// TwinCAT 3 PLC project MPM_PUMP
// ProgramVersion: 3.1.4024.0
// libraries:
//   MPM_FBResult, * (MatrixPM)
//   MPM_JsonParser, * (MatixPM)
//   Tc2_MC2, * (Beckhoff Automation GmbH)
//   Tc2_Standard, * (Beckhoff Automation GmbH)
//   Tc2_System, * (Beckhoff Automation GmbH)
//   Tc2_Utilities, * (Beckhoff Automation GmbH)
//   Tc3_IotBase, * (Beckhoff Automation GmbH)
//   Tc3_Module, * (Beckhoff Automation GmbH)
// project tree:
//   / Class Diagram.TcCD (not stored), PlcTask.TcTTO
//   FBs/Abstracts/ FB_AxisControl.TcPOU, FB_ConfigBase.TcPOU, FB_DiscreteEvents.TcPOU, FB_EventScheduler.TcPOU, FB_PackMLControl.TcPOU, FB_TimeEvents.TcPOU
//   FBs/ FB_EventArray.TcPOU, FB_Kinenmatics.TcPOU, FB_Kinenmatics_V2.TcPOU
//   FBs/IO_Mapping/ FB_IOMappingJson.TcPOU (excluded from build)
//   FBs/IO_Mapping/TcCom/ FB_IOMapping.TcPOU (excluded from build)
//   FBs/IO_Mapping/Types/ ST_IOMappingJson_OLD.TcDUT, ST_IOMappingJson.TcDUT
//   FBs/JSON/ FB_NCAxisJson.TcPOU, FB_NCAxisJson_V2.TcPOU, FB_ValuesJson.TcPOU, ST_AxisMap.TcDUT, ST_AxisMapping.TcDUT
//   FBs/Main/ E_PackMLStates.TcDUT, FB_JsonFile.TcPOU, FB_PackMLControl_Auto.TcPOU, FB_Pump.TcPOU, FB_Squeegee.TcPOU
//   FBs/System/ FB_ConfigControl.TcPOU
//   FUN/ F_Add1.TcPOU, F_INIT_ST_AnyType.TcPOU
//   POUs/ MAIN.TcPOU
// real-time tasks:
//   TASK PlcTask: cycle T#10ms, priority 20, ADS port 350
// motion (NC):
//   TASK NC-Task 1 SAF: cycle T#2ms, priority 4, ADS port 501
//   TASK NC-Task 1 SVB: cycle T#10ms, priority 8, ADS port 511
//   AXIS Axis 1 (id 1)
//     General: UnitName=°
//     Dynamic: Acceleration=5355.76, Deceleration=5355.76, Jerk=16067.3
//     Velo: RefSearch=35.70505, RefSync=35.70505, SlowManual=178.52525, FastManual=1071.1515, Fast=3570.505, Maximum=3570.51
//     OtherSettings: AllowMotionCmdToSlave=true
//     encoder EncType=1
//       EncPara: ScaleFactorNumerator=360, ScaleFactorDenominator=4194304
//     drive DrvType=5
//       Analog: VeloReferenz=3927.5555, TorqueSetpointScale=10, ScaleFactorActTorque=0.1
//       TimeComp: TaskDelayCycles=1
//     controller CtrType=1
//       CtrPara: PriorControlFactor=1
//         Observer: BandWidth=20
// I/O:
//   DEVICE Device 1 (EtherCAT) (disabled), AmsNetId 5.125.204.206.2.1
//     Term 1 (EK1200) [EK1200-5000 EtherCAT Power supply (2A E-Bus)]
//       Term 2 (EL6224) [EL6224 (IO Link Master)]
//       Term 3 (EL1904) [EL1904, 4 Ch. Safety Input 24V, TwinSAFE]
//         modules: Module 1 (FSOES)
//       Term 4 (EL9011) [EL9011 End Terminal]
//   DEVICE Device 2 (EtherCAT) (disabled), AmsNetId 5.125.204.206.3.1
//     Drive 5 (AX5206-0000-0214) [AX5206-0000-0214 EtherCAT Drive (SoE, 2 Ch.)]
// variable links:
//   MPM_PUMP/MPM_PUMP Instance <-> NC-Task 1 SAF/Axes/Axis 1
//     PlcTask Inputs/MAIN.fbPump.axis.NcToPlc <-> Outputs/ToPlc
//     PlcTask Outputs/MAIN.fbPump.axis.PlcToNc <-> Inputs/FromPlc

CONFIGURATION MPM_PUMP
    RESOURCE PLC ON TwinCAT3
        TASK PlcTask(INTERVAL := T#10ms, PRIORITY := 20);
        PROGRAM MAIN WITH PlcTask : MAIN;
    END_RESOURCE
END_CONFIGURATION

// ---- FBs/IO_Mapping/Types/ST_IOMappingJson_OLD.TcDUT
TYPE ST_IOMappingJson_OLD :
STRUCT
	name : STRING;
	deviceNum : WORD;
	channel : USINT;
	ethercatDeviceNum : WORD;
	ioLinkDevice : USINT;
	ioLinkSlaveChannel : USINT;	
	pAny : MPM_JsonParser.ST_AnyType_User;
END_STRUCT
END_TYPE

// ---- FBs/IO_Mapping/Types/ST_IOMappingJson.TcDUT
TYPE ST_IOMappingJson :
STRUCT
	name : STRING;
	deviceNum : WORD;
	channel : USINT;
	ethercatDeviceNum : WORD;
	ioLinkDevice : USINT;
	ioLinkSlaveChannel : USINT;	
	pAny : MPM_JsonParser.ST_AnyType_User;
END_STRUCT
END_TYPE

// ---- FBs/JSON/ST_AxisMap.TcDUT
TYPE ST_AxisMap :
STRUCT
	stAxisMappingJson : ARRAY [0..67] OF  ST_AxisMapping;	
END_STRUCT
END_TYPE

// ---- FBs/JSON/ST_AxisMapping.TcDUT
TYPE ST_AxisMapping :
STRUCT
	name : STRING;
	indexOffset : UDINT;
	pAny : MPM_JsonParser.ST_AnyType_User;
END_STRUCT
END_TYPE

// ---- FBs/Main/E_PackMLStates.TcDUT
{attribute 'qualified_only'}
{attribute 'strict'}
TYPE E_PackMLStates :
(
	idle,
	starting,
	execute,
	completing,
	complete,
	suspdending,
	suspended,
	un_suspsending,
	holding,
	held,
	un_holding,
	aborting,
	aborted,
	stopping,
	stopped
);
END_TYPE

// ---- POUs/MAIN.TcPOU
PROGRAM MAIN
VAR
	ap_fbEvents : ARRAY [0..1023] OF POINTER TO FB_DiscreteEvents; //All assest events combinded
	index : UDINT;
	//machine assets
	fbPump : FB_Pump('fbName');
	fbPump1 : FB_Pump('fbName1');
	fbPump2 : FB_Pump('fbName2');	
	fbPump3 : FB_Pump('fbName3');	
	a_pFBConfigJson : ARRAY [0..3] OF POINTER TO FB_ConfigBase;

	//config control
	fbConfigControl : FB_ConfigControl;
	fbConfigControl_JsonRecipeResult : HRESULT;
	fbConfigControl_JsonSystemResult : HRESULT;
	fbConfigControl_JsonIOResult : HRESULT;
	fbConfigControl_JsonAxisResult : HRESULT;	
	jsonRecipeDoc : STRING(10000);
	jsonSystemDoc : STRING(50000);
	jsonIODoc : STRING(50000);
	jsonAxisDoc : STRING(50000);
	
	//stateMachine
	fbPackMLControlAuto : FB_PackMLControl_Auto; 
	//Node-Red
	fbJsonMQTT : Tc3_IotBase.FB_IotMqttClient;
	mqttPubRate : TON;

END_VAR
//temp 
VAR
	pPointer : ARRAY [0..10] OF POINTER TO MPM_JsonParser.ST_AnyType_User;
	sizeOfValue : DINT;
	position : LREAL;
	dynamicMem : ARRAY [0..65354] OF PVOID;	
	fbKinenmatics : FB_Kinenmatics;
	fbKinenmatics2 : FB_Kinenmatics_V2;	
END_VAR
//Event Test
VAR
x : DINT;
y : DINT;
aLreal : ARRAY [0..0] OF LREAL;
fbPump_OpenValve_Result : HResult := 1;
fbPump_CloseValve_Result : HResult := 1;
fbPump_EnablePump : HResult := 1;
fbPump_HomePump : HResult := 1;
fbPump_MoveAbs : HResult := 1;
fbPump_MoveIncerment : HResult := 1;
fbPump_MoveHalt : HResult := 1;
END_VAR



A_INIT();
A_ConfigControl();
A_Events();

fbPackMLControlAuto.ap_fbEvents := ADR(ap_fbEvents);
fbPackMLControlAuto.M_ExecuteControl();

ACTION A_ConfigControl:


fbConfigControl.a_pFBConfigJson := ADR(a_pFBConfigJson);
fbConfigControl.ua_pFBConfigJson := SIZEOF(a_pFBConfigJson); //Mapping machine assest
//Set json files
fbConfigControl.M_SetJsonRecipe(fbConfigControl_JsonRecipeResult,jsonRecipeDoc);
fbConfigControl.M_SetJsonSystem(fbConfigControl_JsonSystemResult,jsonSystemDoc);
fbConfigControl.M_SetJsonIO(fbConfigControl_JsonIOResult,jsonIODoc);
fbConfigControl.M_SetJsonAxis(fbConfigControl_JsonAxisResult,jsonAxisDoc);
//fbConfigControl_JsonRecipeResult := fbConfigControl.M_GetJsonRecipe(fbConfigControl_JsonRecipeResult,jsonRecipeDoc);


fbJsonMQTT.Execute(TRUE);
mqttPubRate(in := fbJsonMQTT.bConnected, PT := T#500MS);
IF mqttPubRate.Q AND_THEN fbJsonMQTT.Publish('axis',ADR(jsonAxisDoc),LEN2(ADR(jsonAxisDoc)),0,FALSE,FALSE) THEN
	mqttPubRate(in := FALSE);
END_IF
END_ACTION

ACTION A_Events:
fbPump.M_Execute();
fbPump_OpenValve_Result := fbPump.M_Events(fbPump_OpenValve_Result,1);
fbPump_CloseValve_Result := fbPump.M_Events(fbPump_CloseValve_Result,2);
fbPump_EnablePump := fbPump.fbEventEnable.M_Execute(fbPump_EnablePump);
fbPump_HomePump := fbPump.fbEventHomePump.M_Execute(fbPump_HomePump,);
fbPump_MoveIncerment := fbPump.fbEventPumpInterminate.M_Execute(fbPump_MoveIncerment);
fbPump_MoveHalt := fbPump.fbEventMoveHalt.M_Execute(fbPump_MoveHalt);
FOR x := 0 TO 4 BY 1 DO
	fbPump.fbEventMoveAbs.F_GetAnyType(x,p => pPointer[0]);
	F_INIT_ST_AnyType(pPointer[0]);
END_FOR	
fbPump_MoveAbs := fbPump.M_Events(fbPump_MoveAbs,5);

IF fbPump_OpenValve_Result = E_Result.S_OK THEN
	fbPump_OpenValve_Result := E_Result.S_DONE;
END_IF
IF fbPump_CloseValve_Result = E_Result.S_OK THEN
	fbPump_CloseValve_Result := E_Result.S_DONE;
END_IF
IF fbPump_EnablePump = E_Result.S_OK THEN
	fbPump_EnablePump := E_Result.S_DONE;
END_IF
IF fbPump_HomePump = E_Result.S_OK THEN
	fbPump_HomePump := E_Result.S_DONE;
END_IF 
IF fbPump_MoveAbs = E_Result.S_OK THEN
	fbPump_MoveAbs := E_Result.S_DONE;
END_IF 
IF fbPump_MoveIncerment = E_Result.S_OK THEN
	fbPump_MoveIncerment := E_Result.S_DONE;
END_IF 
IF fbPump_MoveHalt = E_Result.S_OK THEN
	fbPump_MoveHalt := E_Result.S_DONE;
END_IF
END_ACTION

ACTION A_INIT:


//Map all 
IF index = 0 THEN
	a_pFBConfigJson[0] := ADR(fbPump);
	a_pFBConfigJson[1] := ADR(fbPump1);
	a_pFBConfigJson[2] := ADR(fbPump2);
	a_pFBConfigJson[3] := ADR(fbPump3);	
	
	FOR x := 0 TO 3 BY 1 DO
		FOR y := 0 TO a_pFBConfigJson[x]^.P_GetNumOfEvents - 1 BY 1 DO
			IF a_pFBConfigJson[x]^.M_GetEvent(ADR(ap_fbEvents[index]),y) = E_Result.S_OK THEN
				index := index + 1;	
			ELSE
				CONTINUE;
			END_IF	
		END_FOR
	END_FOR
END_IF
END_ACTION

END_PROGRAM

// ---- FBs/Abstracts/FB_DiscreteEvents.TcPOU
(*
Standard way to set up events to be tied to other parts of the project. might make an interface
*)
{attribute 'reflection'} 
FUNCTION_BLOCK FB_DiscreteEvents
VAR_INPUT
END_VAR
VAR_OUTPUT
END_VAR
VAR
	pstAnyType_User : POINTER TO MPM_JsonParser.ST_AnyType_User; //array 
	uAnyType_User : DINT; //Len of array 
	pfbConfigBase : POINTER TO FB_ConfigBase; 
	eventID : DINT;
    {attribute 'instance-path'} 
    {attribute 'noinit'}	
	_eventName : STRING(1024);
END_VAR
VAR CONSTANT
	sizeOfAnyType_User : DINT := SIZEOF(MPM_JsonParser.ST_AnyType_User);
END_VAR

METHOD PUBLIC F_GetAnyType : HResult
VAR_INPUT
	arrayPosition : DINT;
END_VAR
VAR_OUTPUT
	p : POINTER TO MPM_JsonParser.ST_AnyType_User;
END_VAR
VAR
	pointerOffset : DINT;
END_VAR
IF pstAnyType_User = 0 THEN // no values
	F_GetAnyType := MPM_FBResult.E_Result.S_FAILED;
END_IF
F_GetAnyType := pfbConfigBase^.F_GetArrayPosition(uAnyType_User,sizeOfAnyType_User,arrayPosition,offset => pointerOffset);
IF F_GetAnyType = MPM_FBResult.E_Result.S_OK THEN
	p := pstAnyType_User + pointerOffset;
ELSE
	F_GetAnyType := MPM_FBResult.E_Result.S_FAILED;
END_IF
END_METHOD

METHOD FB_exit : BOOL
VAR_INPUT
	bInCopyCode : BOOL; // if TRUE, the exit method is called for exiting an instance that is copied afterwards (online change).
END_VAR

VAR
	pstAnyType_User : POINTER TO MPM_JsonParser.ST_AnyType_User; //array 
	length : DINT; 
	offset : DINT;
	x : DINT;
	pByte : POINTER TO BYTE;
END_VAR
IF bInCopyCode = FALSE THEN
	IF pfbConfigBase^.F_GetArrayLength(uAnyType_User,sizeOfAnyType_User, length => length) = MPM_FBResult.E_Result.S_OK THEN
		FOR x := 0 TO length BY 1 DO
			pfbConfigBase^.F_GetArrayPosition(uAnyType_User,sizeOfAnyType_User,x,offset => offset);
			pstAnyType_User := THIS^.pstAnyType_User + offset;
			pByte := pstAnyType_User^.pvalue;
			__DELETE(pByte);
		END_FOR
	END_IF
END_IF
END_METHOD

METHOD FB_init : BOOL
VAR_INPUT
	bInitRetains : BOOL; // if TRUE, the retain variables are initialized (warm start / cold start)
	bInCopyCode : BOOL;  // if TRUE, the instance afterwards gets moved into the copy code (online change)
	pfbConfigBase : POINTER TO FB_ConfigBase; 
	eventID : DINT;
	pstAnyType_User : POINTER TO MPM_JsonParser.ST_AnyType_User; //array 
	uAnyType_User : DINT; //Len of array 	
END_VAR
THIS^.pfbConfigBase := pfbConfigBase;
THIS^.pstAnyType_User := pstAnyType_User;
THIS^.uAnyType_User := uAnyType_User;
THIS^.eventID := eventID;
END_METHOD

METHOD PUBLIC M_Execute : HRESULT
VAR_INPUT
	lastResult : HResult;
END_VAR
IF pfbConfigBase > 0 THEN 
	M_Execute := pfbConfigBase^.M_Events(lastResult,eventID);
END_IF
END_METHOD

PROPERTY PUBLIC P_EventId : Dint
GET
END_GET
END_PROPERTY

PROPERTY PUBLIC P_EventName : String(1024)
GET
P_EventName := _eventName;
END_GET
END_PROPERTY

END_FUNCTION_BLOCK

// ---- FBs/Abstracts/FB_ConfigBase.TcPOU
(*
Will be an abstract class that will be used to configure all parts of the machine through json
*)

FUNCTION_BLOCK ABSTRACT FB_ConfigBase
VAR_INPUT
END_VAR
VAR_OUTPUT
END_VAR
VAR 
	_fbName : STRING; //name of FB set on init
END_VAR

METHOD _F_Axis : HRESULT
VAR_IN_OUT
	a_pstAxisParameterSet : POINTER TO Tc2_MC2.ST_AxisParameterSet; //pointer to array
	pstAxisMapping : UDINT;
END_VAR
END_METHOD

METHOD PROTECTED ABSTRACT _F_IO : HResult
VAR_IN_OUT
	a_pstIOMappingJson : POINTER TO ST_IOMappingJson; //pointer to array
	ustIOMappingJson : UDINT; 		
END_VAR
END_METHOD

(*
return the list of vars that want to be saved and loaded 
*)

METHOD PROTECTED ABSTRACT _F_Recipe : HResult
VAR_IN_OUT
	a_pstAnyTypeUser : POINTER TO MPM_JsonParser.ST_AnyType_User; //pointer to array
	uAnyTypeUser : UDINT; //size of array	
END_VAR
VAR_OUTPUT

END_VAR
END_METHOD

METHOD PROTECTED ABSTRACT _F_System : HResult
VAR_IN_OUT
	a_pstAnyTypeUser : POINTER TO MPM_JsonParser.ST_AnyType_User; //pointer to array
	uAnyTypeUser : UDINT; //size of array	
END_VAR
END_METHOD

METHOD PUBLIC FINAL F_AXIS : HRESULT
VAR_INPUT
	lastResult : HRESULT;
	sJson : SJsonValue;
	pfbJsonSchema : POINTER TO FB_NCAxisJson_V2;	
	bGet : BOOL;
END_VAR

VAR_INST
	_fbResult : FB_ResultHelper_V2;
	pResult : POINTER TO HRESULT;
END_VAR

VAR
	a_pstAxisParameterSet : POINTER TO Tc2_MC2.ST_AxisParameterSet;
	dstAxisParameterSet : UDINT; //number of bytes in a_stAnyUser
	
	uSizeOfArray : UDINT;
	
	pstAxisParameterSet : POINTER TO Tc2_MC2.ST_AxisParameterSet; //pointer for loop
	x : UDINT;
END_VAR


VAR CONSTANT
	uSizeOfStAnyType : UDINT := SIZEOF(Tc2_MC2.ST_AxisParameterSet);
END_VAR
IF _fbResult.M_MethodResult(F_AXIS,ADR(pResult),lastResult) = FALSE THEN
	RETURN;
END_IF


pResult^ := _F_Axis(a_pstAxisParameterSet,dstAxisParameterSet);
//pResult^ := MPM_FBResult.E_Result.S_WORKING;
IF bGet = FALSE THEN
	sJson := pfbJsonSchema^.M_SetJsonMember(sJson,_fbName);
	IF a_pstAxisParameterSet > 0 AND dstAxisParameterSet > 0 AND uSizeOfStAnyType > 0 THEN //make sure all values are vaild
		uSizeOfArray := dstAxisParameterSet/uSizeOfStAnyType - 1; //get number of items in array
		FOR x := 0 TO uSizeOfArray BY 1 DO //loop through all items 
			pstAxisParameterSet := a_pstAxisParameterSet + uSizeOfStAnyType*x; // get array position
			pResult^ := pfbJsonSchema^.M_SetAxisJson(pResult^,sJson,pstAxisParameterSet);
		END_FOR
	END_IF	
ELSIF bGet = TRUE THEN
	sJson := pfbJsonSchema^.FindMember(sJson,_fbName);
	IF a_pstAxisParameterSet > 0 AND dstAxisParameterSet > 0 AND uSizeOfStAnyType > 0 THEN //make sure all values are vaild
		uSizeOfArray := dstAxisParameterSet/uSizeOfStAnyType - 1; //get number of items in array
		FOR x := 0 TO uSizeOfArray BY 1 DO //loop through all items 
			pstAxisParameterSet := a_pstAxisParameterSet + uSizeOfStAnyType*x; // get array position
			pResult^ := pfbJsonSchema^.M_GetAxisJson(pResult^,sJson,pstAxisParameterSet);
		END_FOR
	END_IF
END_IF
END_METHOD

METHOD PROTECTED F_Event_ST_AnyType_Compare : HResult
VAR_INPUT
	srcvar : POINTER TO MPM_JsonParser.ST_AnyType_User; //PVOID FOR any value
	desvar : POINTER TO MPM_JsonParser.ST_AnyType_User;	//What was input
END_VAR
VAR
END_VAR
IF srcvar^.typeclass = desvar^.typeclass AND srcvar^.diSize = desvar^.diSize THEN
	desvar^.pvalue := srcvar^.pvalue;
	F_Event_ST_AnyType_Compare := MPM_FBResult.E_Result.S_OK;
ELSE
	F_Event_ST_AnyType_Compare := MPM_FBResult.E_Result.S_FAILED;	
END_IF
END_METHOD

METHOD PUBLIC F_GetArrayLength : HResult
VAR_INPUT
	sizeOfInst : DINT;
	sizeOFType : DINT;
END_VAR
VAR_OUTPUT
	length : DINT;
END_VAR
VAR
	_numOfElements : DINT;
END_VAR
IF sizeOFType > 0 AND sizeOfInst > 0 THEN
	_numOfElements := sizeOfInst/sizeOFType -1;
	IF _numOfElements > 0 THEN
		length := _numOfElements;
		F_GetArrayLength := MPM_FBResult.E_Result.S_OK;
	END_IF
ELSE
	F_GetArrayLength := MPM_FBResult.E_Result.S_FAILED;
	RETURN;
END_IF
END_METHOD

METHOD PUBLIC F_GetArrayPosition : HResult
VAR_INPUT
	sizeOfInst : DINT;
	sizeOFType : DINT;
	index : DINT;
END_VAR
VAR_OUTPUT
	offset : DINT;
	length : DINT;
END_VAR
VAR
END_VAR
F_GetArrayPosition := F_GetArrayLength(sizeOfInst,sizeOFType, length => length);
IF F_GetArrayPosition = MPM_FBResult.E_Result.S_OK THEN
	IF index >= 0 AND index <= length THEN
		offset := sizeOFType*index;
	ELSE
		F_GetArrayPosition := MPM_FBResult.E_Result.S_FAILED;
	END_IF
ELSE
	F_GetArrayPosition := MPM_FBResult.E_Result.S_OK;
END_IF
END_METHOD

METHOD PUBLIC FINAL F_IO : HRESULT
VAR_INPUT
	lastResult : HRESULT;
	sJson : SJsonValue;
	pfbJsonSchema : POINTER TO FB_JsonSchemaEx_OLD;
	bGet : BOOL;	
END_VAR

VAR_INST
	_fbResult : FB_ResultHelper_V2;
	pResult : POINTER TO HRESULT;
END_VAR

VAR
	a_pstIOMappingJson : POINTER TO ST_IOMappingJson; // pointer to array of vars
	uAnyTypeUser : UDINT; //number of bytes in a_stAnyUser
	
	uSizeOfArray : UDINT;
	pstIOMappingJson : POINTER TO ST_IOMappingJson; //pointer for loop
	x : UDINT;
END_VAR


VAR CONSTANT
	uSizeOfStAnyType : UDINT := SIZEOF(ST_IOMappingJson);
END_VAR
IF _fbResult.M_MethodResult(F_IO,ADR(pResult),lastResult) = FALSE THEN
	RETURN;
END_IF


pResult^ := _F_IO(a_pstIOMappingJson,uAnyTypeUser); //gets pointer from FB


pResult^ := MPM_FBResult.E_Result.S_WORKING;
//set
IF bGet = FALSE THEN
	sJson := pfbJsonSchema^.M_SetJsonMember(sJson,_fbName);
	IF a_pstIOMappingJson > 0 AND_THEN uAnyTypeUser > 0 AND uSizeOfStAnyType > 0 THEN //make sure all values are vaild
		uSizeOfArray := uAnyTypeUser/uSizeOfStAnyType - 1; //get number of items in array
		FOR x := 0 TO uSizeOfArray BY 1 DO //loop through all items 
			pstIOMappingJson := a_pstIOMappingJson + uSizeOfStAnyType*x; // get array position
			sJson := pfbJsonSchema^.M_SetJsonMember(sJson,pstIOMappingJson^.name); //set json value
			pfbJsonSchema^.M_SetJsonMemberValue(sJson,'deviceNum',pstIOMappingJson^.deviceNum); //set json value			
			pfbJsonSchema^.M_SetJsonMemberValue(sJson,'channel',pstIOMappingJson^.channel); //set json value
			//IO-link
			pfbJsonSchema^.M_SetJsonMemberValue(sJson,'ethercatDeviceNum',pstIOMappingJson^.ethercatDeviceNum); //set json value
			pfbJsonSchema^.M_SetJsonMemberValue(sJson,'ioLinkDevice',pstIOMappingJson^.ioLinkDevice); //set json value
			pfbJsonSchema^.M_SetJsonMemberValue(sJson,'ioLinkSlaveChannel',pstIOMappingJson^.ioLinkSlaveChannel); //set json value
		END_FOR
		pResult^ := MPM_FBResult.E_Result.S_OK;
	ELSE
		pResult^ := MPM_FBResult.E_Result.S_FAILED;
	END_IF
//get
ELSIF bGet = TRUE THEN
	sJson := pfbJsonSchema^.FindMember(sJson,_fbName);
	IF a_pstIOMappingJson > 0 AND_THEN uAnyTypeUser > 0 AND uSizeOfStAnyType > 0 THEN //make sure all values are vaild
		uSizeOfArray := uAnyTypeUser/uSizeOfStAnyType - 1; //get number of items in array
		FOR x := 0 TO uSizeOfArray BY 1 DO //loop through all items 
			pstIOMappingJson := a_pstIOMappingJson + uSizeOfStAnyType*x; // get array position
			sJson := pfbJsonSchema^.M_SetJsonMember(sJson,pstIOMappingJson^.name); //set json value
			pfbJsonSchema^.M_GetJsonMemberValue(sJson,'channel',pstIOMappingJson^.channel); //set json value
			pfbJsonSchema^.M_GetJsonMemberValue(sJson,'deviceNum',pstIOMappingJson^.deviceNum); //set json value
			pfbJsonSchema^.M_GetJsonMemberValue(sJson,'ethercatDeviceNum',pstIOMappingJson^.ethercatDeviceNum); //set json value
			pfbJsonSchema^.M_GetJsonMemberValue(sJson,'ioLinkDevice',pstIOMappingJson^.ioLinkDevice); //set json value
			pfbJsonSchema^.M_GetJsonMemberValue(sJson,'ioLinkSlaveChannel',pstIOMappingJson^.ioLinkSlaveChannel); //set json value
		END_FOR
		pResult^ := MPM_FBResult.E_Result.S_OK;
	ELSE
		pResult^ := MPM_FBResult.E_Result.S_FAILED;
	END_IF
END_IF
END_METHOD

METHOD PROTECTED F_Map_ST_IOMappingJson : HRESULT
VAR_INPUT
	stIOMappingJson : POINTER TO ST_IOMappingJson;
	name : STRING;
	pPVoid : POINTER TO PVOID;
END_VAR
END_METHOD

METHOD PUBLIC FINAL F_Recipe : HRESULT
VAR_INPUT
	lastResult : HRESULT;
	sJson : SJsonValue;
	pfbJsonSchema : POINTER TO FB_JsonSchemaEx_OLD;	
	bGet : BOOL;
END_VAR

VAR_INST
	_fbResult : FB_ResultHelper_V2;
	pResult : POINTER TO HRESULT;
END_VAR

VAR
	a_stAnyUser : POINTER TO MPM_JsonParser.ST_AnyType_User; // pointer to array of vars
	uAnyTypeUser : UDINT; //number of bytes in a_stAnyUser
	
	uSizeOfArray : UDINT;
	pstAnyUser : POINTER TO MPM_JsonParser.ST_AnyType_User; //pointer for loop
	x : UDINT;
END_VAR

VAR CONSTANT
	uSizeOfStAnyType : UDINT := SIZEOF(MPM_JsonParser.ST_AnyType_User);
END_VAR
IF _fbResult.M_MethodResult(F_Recipe,ADR(pResult),lastResult) = FALSE THEN
	RETURN;
END_IF


pResult^ := _F_Recipe(a_stAnyUser,uAnyTypeUser);


pResult^ := MPM_FBResult.E_Result.S_WORKING;

//set
IF bGet = FALSE THEN
	sJson := pfbJsonSchema^.M_SetJsonMember(sJson,_fbName);
	IF a_stAnyUser > 0 AND_THEN uAnyTypeUser > 0 AND uSizeOfStAnyType > 0 THEN //make sure all values are vaild
		uSizeOfArray := uAnyTypeUser/uSizeOfStAnyType - 1; //get number of items in array
		FOR x := 0 TO uSizeOfArray BY 1 DO //loop through all items 
			pstAnyUser := a_stAnyUser + uSizeOfStAnyType*x; // get array position
				pfbJsonSchema^.M_SetJsonMemberValue_AnyType(sJson,pstAnyUser^.name,pstAnyUser^); //set json value
		END_FOR
		pResult^ := MPM_FBResult.E_Result.S_OK;
	ELSE
		pResult^ := MPM_FBResult.E_Result.S_FAILED;
	END_IF
	
//get
ELSIF bGet = TRUE THEN 	
	sJson := pfbJsonSchema^.FindMember(sJson,_fbName);
	IF a_stAnyUser > 0 AND_THEN uAnyTypeUser > 0 AND uSizeOfStAnyType > 0 THEN //make sure all values are vaild
		uSizeOfArray := uAnyTypeUser/uSizeOfStAnyType - 1; //get number of items in array
		FOR x := 0 TO uSizeOfArray BY 1 DO //loop through all items 
			pstAnyUser := a_stAnyUser + uSizeOfStAnyType*x; // get array position
				pfbJsonSchema^.M_GetJsonMemberValue_AnyType(sJson,pstAnyUser^.name,pstAnyUser^); //set json value
		END_FOR
		pResult^ := MPM_FBResult.E_Result.S_OK;
	ELSE
		pResult^ := MPM_FBResult.E_Result.S_FAILED;
	END_IF
END_IF
END_METHOD

METHOD PUBLIC FINAL F_System : HRESULT
VAR_INPUT
	lastResult : HRESULT;
	sJson : SJsonValue;
	pfbJsonSchema : POINTER TO FB_JsonSchemaEx_OLD;	
	bGet : BOOL;	
END_VAR

VAR_INST
	_fbResult : FB_ResultHelper_V2;
	pResult : POINTER TO HRESULT;
END_VAR

VAR
	a_stAnyUser : POINTER TO MPM_JsonParser.ST_AnyType_User; // pointer to array of vars
	uAnyTypeUser : UDINT; //number of bytes in a_stAnyUser
	
	uSizeOfArray : UDINT;
	pstAnyUser : POINTER TO MPM_JsonParser.ST_AnyType_User; //pointer for loop
	x : UDINT;
END_VAR


VAR CONSTANT
	uSizeOfStAnyType : UDINT := SIZEOF(MPM_JsonParser.ST_AnyType_User);
END_VAR
IF _fbResult.M_MethodResult(F_System,ADR(pResult),lastResult) = FALSE THEN
	RETURN;
END_IF


pResult^ := _F_System(a_stAnyUser,uAnyTypeUser);
//set
IF bGet = FALSE THEN
	pResult^ := MPM_FBResult.E_Result.S_WORKING;
	sJson := pfbJsonSchema^.M_SetJsonMember(sJson,_fbName);
	IF a_stAnyUser > 0 AND_THEN uAnyTypeUser > 0 AND uSizeOfStAnyType > 0 THEN //make sure all values are vaild
		uSizeOfArray := uAnyTypeUser/uSizeOfStAnyType - 1; //get number of items in array
		FOR x := 0 TO uSizeOfArray BY 1 DO //loop through all items 
			pstAnyUser := a_stAnyUser + uSizeOfStAnyType*x; // get array position
				pfbJsonSchema^.M_SetJsonMemberValue_AnyType(sJson,pstAnyUser^.name,pstAnyUser^); //set json value
		END_FOR
		pResult^ := MPM_FBResult.E_Result.S_OK;
	ELSE
		pResult^ := MPM_FBResult.E_Result.S_FAILED;
	END_IF

//get	
ELSIF bGet = TRUE THEN
	sJson := pfbJsonSchema^.FindMember(sJson,_fbName);
	IF a_stAnyUser > 0 AND_THEN uAnyTypeUser > 0 AND uSizeOfStAnyType > 0 THEN //make sure all values are vaild
		uSizeOfArray := uAnyTypeUser/uSizeOfStAnyType - 1; //get number of items in array
		FOR x := 0 TO uSizeOfArray BY 1 DO //loop through all items 
			pstAnyUser := a_stAnyUser + uSizeOfStAnyType*x; // get array position
				pfbJsonSchema^.M_GetJsonMemberValue_AnyType(sJson,pstAnyUser^.name,pstAnyUser^); //set json value
		END_FOR
		pResult^ := MPM_FBResult.E_Result.S_OK;
	ELSE
		pResult^ := MPM_FBResult.E_Result.S_FAILED;
	END_IF	
END_IF
END_METHOD

METHOD PROTECTED F_TO_LREAL : LREAL
VAR_INPUT
	pPvoid : PVOID;
END_VAR
VAR_OUTPUT
	error : BOOL;
END_VAR
VAR
	pLREAL : POINTER TO LREAL;
END_VAR
IF pPvoid > 0 THEN
	pLREAL := pPvoid;
	F_TO_LREAL := pLREAL^;
ELSE
	error := TRUE;
END_IF
END_METHOD

METHOD FB_init : BOOL
VAR_INPUT
	bInitRetains : BOOL; // if TRUE, the retain variables are initialized (warm start / cold start)
	bInCopyCode : BOOL;  // if TRUE, the instance afterwards gets moved into the copy code (online change)
	fbName : STRING;
END_VAR
_fbName := fbName;
END_METHOD

METHOD PUBLIC ABSTRACT M_Events : HResult
VAR_INPUT
	lastResult : HResult;
	eventID : DINT;
END_VAR
END_METHOD

METHOD PUBLIC ABSTRACT M_Execute : HRESULT
VAR_INPUT
END_VAR
VAR_INST

END_VAR
END_METHOD

METHOD PUBLIC ABSTRACT M_GetEvent : HResult
VAR_INPUT
	pFbDiscreteEvents : POINTER TO POINTER TO FB_DiscreteEvents;
	index : DINT;	
END_VAR
END_METHOD

PROPERTY PUBLIC P_fbName : STRING
GET
P_fbName := _fbName;
END_GET
END_PROPERTY

PROPERTY PUBLIC ABSTRACT P_GetNumOfEvents : DINT
GET
END_GET
END_PROPERTY

END_FUNCTION_BLOCK

// ---- FBs/JSON/FB_NCAxisJson_V2.TcPOU
{attribute 'call_after_init'}
FUNCTION_BLOCK FB_NCAxisJson_V2 EXTENDS FB_JsonSchemaEx_OLD
VAR_INPUT
		
END_VAR
VAR_OUTPUT
	P_sJsonid			: MPM_JsonParser.DUT_JsonSchema := (member := '_id', typeClass := E_TypeClassEx.TYPE_STRING,jsonValueRoot := jsonRoot);
	P_sJsonTimeStamp	: MPM_JsonParser.DUT_JsonSchema := (member := 'time_stamp', typeClass := E_TypeClassEx.TYPE_FILETIME,jsonValueRoot := jsonRoot);		
	P_sJsonValues		: MPM_JsonParser.DUT_JsonSchema := (member := 'values', typeClass := E_TypeClassEx.TYPE_JSON,jsonValueRoot := jsonRoot);
END_VAR
VAR
	jsonRoot : SJsonValue;
	adsRead : ADSReadEX;
	saveTemplete : BOOL := FALSE;
	stAxisMappingJson : ST_AxisMap;
END_VAR
VAR_OUTPUT
	//stIOMappingEthercat : ARRAY [0..NUM_OF_VARS] OF ST_IOMappingEthercatJson;	
END_VAR
VAR CONSTANT
	NUM_OF_VARS : DINT :=  67;
	INDEX_BASE : DINT :=  16384;
	PORT : UINT := 501;
END_VAR

METHOD PROTECTED _M_MapJsonValues : HRESULT
VAR_INPUT
	stAxisMappingJson : REFERENCE TO ST_AxisMapping;
	name : STRING;
	indexOffset : UDINT;
	pAny : ANY;
END_VAR
stAxisMappingJson.name := name;
stAxisMappingJson.indexOffset := indexOffset;
stAxisMappingJson.pAny.typeclass := TO_INT(pAny.TypeClass);
stAxisMappingJson.pAny.pvalue := pAny.pValue;
stAxisMappingJson.pAny.diSize := pAny.diSize;
END_METHOD

METHOD PUBLIC  M_CreateSchemaJson : BOOL
VAR_IN_OUT
END_VAR
VAR
	
END_VAR
jsonRoot := THIS^.NewDocument();
M_SetJsonSchema(jsonRoot,P_sJsonid);
//M_SetJsonSchema(P_sJsonid.jsonValue,P_sJsonRecipe);
M_SetJsonSchema(jsonRoot,P_sJsonValues);
M_SetJsonSchema(jsonRoot,P_sJsonTimeStamp);
END_METHOD

METHOD PUBLIC M_GetAxisJson : HRESULT
VAR_INPUT
	lastResult : HRESULT;
	pJson : SJsonValue;	
END_VAR
VAR_INPUT
	pAxisParamters : POINTER TO Tc2_MC2.ST_AxisParameterSet;
END_VAR
VAR_INST
	loadFile : BOOL;		
	x : UDINT;
	aStringJson : STRING(10000);
	fileName : STRING(255);
	_state			: DINT;
	_fbResult		: FB_ResultHelper;	
	errorCode : HRESULT;
END_VAR

VAR

END_VAR
IF _fbResult.M_MethodResult(M_GetAxisJson,lastResult) = FALSE THEN
	RETURN;
ELSE

	IF _fbResult.P_Result = E_Result.S_OK THEN //Reset
		_state := 0;	
		x := 0;
	END_IF 

	_fbResult.P_Result := E_Result.S_WORKING; //Working	
	
	CASE _state OF
		0:
			FOR x := 0 TO NUM_OF_VARS BY 1 DO
				pJson := THIS^.FindMember(P_sJsonValues.jsonValue,stAxisMappingJson.stAxisMappingJson[x].name);	
				IF pJson > 0 THEN
					THIS^.M_GetAxisJson_Values(pJson,ADR(stAxisMappingJson.stAxisMappingJson[x]),pAxisParamters);
				END_IF	
			END_FOR	
			_fbResult.P_Result := E_Result.S_OK; //OK				
		END_CASE
END_IF
END_METHOD

METHOD PROTECTED M_GetAxisJson_Values : HResult
VAR_INPUT
	sJson : SJsonValue;
	stAxisMapping : POINTER TO ST_AxisMapping;
	pAxisParamters : POINTER TO Tc2_MC2.ST_AxisParameterSet;	
END_VAR

VAR
	pAny : MPM_JsonParser.ST_AnyType_User;	
END_VAR
pAny := stAxisMapping^.pAny;
pAny.pvalue := pAny.pvalue + pAxisParamters;
THIS^.M_GetJsonMemberValue_AnyType(sJson,'value',pAny);
END_METHOD

METHOD PUBLIC M_GetParametersFromAxis : HResult
VAR_INPUT
	lastResult : HRESULT;
	axisID : DINT;
	pAxisParamters : POINTER TO Tc2_Mc2.ST_AxisParameterSet;
END_VAR	


VAR_INST
	adsRead : ADSRead;	
	_state			: DINT;
	_fbResult		: FB_ResultHelper;
	x : DINT;
END_VAR
IF _fbResult.M_MethodResult(M_GetParametersFromAxis,lastResult) = FALSE THEN
	RETURN;
ELSE
	
	IF _fbResult.P_Result = E_Result.S_OK THEN //Reset
		_state := 0;	
		adsRead(READ := FALSE);
		x := 0;
	END_IF 
	
	_fbResult.P_Result := E_Result.S_WORKING; //Working	
	
	CASE _state OF
		0:
			adsRead.port := PORT;
			adsRead.IDXGRP := INDEX_BASE + axisID;
			adsRead.IDXOFFS :=stAxisMappingJson[x].indexOffset;
			adsRead.LEN := stAxisMappingJson[x].pAny.diSize;
			adsRead.DESTADDR := stAxisMappingJson[x].pAny.pvalue + pAxisParamters; //very important how this works
			adsRead(READ := TRUE);
			_state := 1;
		1:
			adsRead(READ := TRUE);
			IF adsRead.READ = TRUE AND adsRead.BUSY = FALSE AND adsRead.ERR = FALSE THEN
				IF x < NUM_OF_VARS THEN
					x := x + 1;
					adsRead(READ := FALSE);
					_state := 0;
				ELSIF x >= NUM_OF_VARS THEN
					_fbResult.P_Result := E_Result.S_OK;
				END_IF
			ELSIF adsRead.READ = TRUE AND adsRead.BUSY = FALSE AND adsRead.ERR = TRUE THEN
				ADSLOGSTR(msgCtrlMask := ADSLOG_MSGTYPE_ERROR,
					msgFmtStr := 'Error in %s',
					strArg := stAxisMappingJson[x].name);
				ADSLOGSTR(msgCtrlMask := ADSLOG_MSGTYPE_ERROR,
					msgFmtStr := 'ErrorID %s',
					strArg := TO_STRING(adsRead.ERRID));
				_fbResult.P_Result := E_Result.S_FAILED;	
			END_IF	
	END_CASE
END_IF
END_METHOD

{attribute 'call_after_init'}
METHOD PROTECTED M_MapJsonValues : HResult
VAR_INPUT
END_VAR
VAR
	x : DINT;
	pAxisParamters : POINTER TO TC2_MC2.ST_AxisParameterSet;;	
END_VAR
(* AXIS: *)
_M_MapJsonValues(stAxisMappingJson.stAxisMappingJson[F_Add1(x)],'AxisId',16#1,pAxisParamters^.AxisId); // AxisId                      : DWORD; (* 0x00000001 *)
_M_MapJsonValues(stAxisMappingJson.stAxisMappingJson[F_Add1(x)],'sAxisName',16#2,pAxisParamters^.sAxisName);// sAxisName                   : STRING(31); (* 0x00000002 *)
_M_MapJsonValues(stAxisMappingJson.stAxisMappingJson[F_Add1(x)],'nAxisType',16#3,pAxisParamters^.nAxisType); // nAxisType                   : DWORD;      (* 0x00000003 *)
_M_MapJsonValues(stAxisMappingJson.stAxisMappingJson[F_Add1(x)],'bEnablePositionAreaControl',16#F,pAxisParamters^.bEnablePositionAreaControl);// bEnablePositionAreaControl  : WORD;       (* 0x0000000F *)
_M_MapJsonValues(stAxisMappingJson.stAxisMappingJson[F_Add1(x)],'fPositionAreaControlRange',16#10,pAxisParamters^.fPositionAreaControlRange);// fPositionAreaControlRange   : LREAL;      (* 0x00000010 *)
_M_MapJsonValues(stAxisMappingJson.stAxisMappingJson[F_Add1(x)],'bEnableMotionControl',16#11,pAxisParamters^.bEnableMotionControl);// bEnableMotionControl        : WORD;       (* 0x00000011 *)
_M_MapJsonValues(stAxisMappingJson.stAxisMappingJson[F_Add1(x)],'fMotionControlTime',16#12,pAxisParamters^.fMotionControlTime);// fMotionControlTime          : LREAL;      (* 0x00000012 *)
_M_MapJsonValues(stAxisMappingJson.stAxisMappingJson[F_Add1(x)],'bEnableLoop',16#13,pAxisParamters^.bEnableLoop);//   bEnableLoop                 : WORD;       (* 0x00000013 *)
_M_MapJsonValues(stAxisMappingJson.stAxisMappingJson[F_Add1(x)],'fLoopDistance',16#14,pAxisParamters^.fLoopDistance);// fLoopDistance               : LREAL;      (* 0x00000014 *)
_M_MapJsonValues(stAxisMappingJson.stAxisMappingJson[F_Add1(x)],'bEnableTargetPosControl',16#15,pAxisParamters^.bEnableTargetPosControl);// bEnableTargetPosControl     : WORD;       (* 0x00000015 *)
_M_MapJsonValues(stAxisMappingJson.stAxisMappingJson[F_Add1(x)],'fTargetPosControlRange',16#16,pAxisParamters^.fTargetPosControlRange);// fTargetPosControlRange      : LREAL;      (* 0x00000016 *)
_M_MapJsonValues(stAxisMappingJson.stAxisMappingJson[F_Add1(x)],'fTargetPosControlTime',16#17,pAxisParamters^.fTargetPosControlTime);// fTargetPosControlTime       : LREAL;      (* 0x00000017 *)
_M_MapJsonValues(stAxisMappingJson.stAxisMappingJson[F_Add1(x)],'fVeloMaximum',16#27,pAxisParamters^.fVeloMaximum);// fVeloMaximum                : LREAL;      (* 0x00000027 *)
_M_MapJsonValues(stAxisMappingJson.stAxisMappingJson[F_Add1(x)],'fMotionControlRange',16#28,pAxisParamters^.fMotionControlRange);// fMotionControlRange         : LREAL;      (* 0x00000028 *)
_M_MapJsonValues(stAxisMappingJson.stAxisMappingJson[F_Add1(x)],'bEnablePEHTimeControl',16#29,pAxisParamters^.bEnablePEHTimeControl);// bEnablePEHTimeControl       : WORD;       (* 0x00000029 *)
_M_MapJsonValues(stAxisMappingJson.stAxisMappingJson[F_Add1(x)],'fPEHControlTime',16#2A,pAxisParamters^.fPEHControlTime);// fPEHControlTime             : LREAL;      (* 0x0000002A *)
_M_MapJsonValues(stAxisMappingJson.stAxisMappingJson[F_Add1(x)],'bEnableBacklashCompensation',16#2B,pAxisParamters^.bEnableBacklashCompensation);// bEnableBacklashCompensation : WORD;       (* 0x0000002B *)
_M_MapJsonValues(stAxisMappingJson.stAxisMappingJson[F_Add1(x)],'fBacklash',16#2C,pAxisParamters^.fBacklash);// fBacklash                   : LREAL;      (* 0x0000002C *))
//_M_MapJsonValues(stAxisMappingJson[F_Add1(x)],'sAmsNetId',16#31,pAxisParamters^.sAmsNetId);// sAmsNetId : WORD;       (* 0x00000031 *)
//_M_MapJsonValues(stAxisMappingJson[F_Add1(x)],'nPort',16#31,pAxisParamters^.nPort);// nPort : WORD;       (* 0x00000031 *)*)
//_M_MapJsonValues(stAxisMappingJson[F_Add1(x)],'fDeceleration',16#102,pAxisParamters^.fDeceleration);//fDeceleration               : LREAL;      (* 0x00000101
//_M_MapJsonValues(stAxisMappingJson[F_Add1(x)],'nChnNo',16#31,pAxisParamters^.nChnNo);// nChnNo : WORD;       (* 0x00000031 *)
_M_MapJsonValues(stAxisMappingJson.stAxisMappingJson[F_Add1(x)],'fAcceleration',16#101,pAxisParamters^.fAcceleration);//fAcceleration               : LREAL;      (* 0x00000101 *)
_M_MapJsonValues(stAxisMappingJson.stAxisMappingJson[F_Add1(x)],'fDeceleration',16#102,pAxisParamters^.fDeceleration);//fDeceleration               : LREAL;      (* 0x00000102  *)
_M_MapJsonValues(stAxisMappingJson.stAxisMappingJson[F_Add1(x)],'fAccelerationMax',16#F1,pAxisParamters^.fAccelerationMax);//fAcceleration               : LREAL;      (* 0x00000101 *)
_M_MapJsonValues(stAxisMappingJson.stAxisMappingJson[F_Add1(x)],'fDecelerationMax',16#F2,pAxisParamters^.fDecelerationMax);//fDeceleration               : LREAL;      (* 0x00000102  *)
_M_MapJsonValues(stAxisMappingJson.stAxisMappingJson[F_Add1(x)],'fJerk',16#103,pAxisParamters^.fJerk);//fJerk                       : LREAL;      (* 0x00000103 *)
(* ENCODER: *)
_M_MapJsonValues(stAxisMappingJson.stAxisMappingJson[F_Add1(x)],'nEncId',16#10001,pAxisParamters^.nEncId);//nEncId                      : DWORD;      (* 0x00010001 *)
_M_MapJsonValues(stAxisMappingJson.stAxisMappingJson[F_Add1(x)],'sEncName',16#10002,pAxisParamters^.sEncName);//sEncName                    : STRING(31); (* 0x00010002 *)
_M_MapJsonValues(stAxisMappingJson.stAxisMappingJson[F_Add1(x)],'nEncType',16#10003,pAxisParamters^.nEncType);//nEncType                    : DWORD;      (* 0x00010003 *)
_M_MapJsonValues(stAxisMappingJson.stAxisMappingJson[F_Add1(x)],'fEncScaleFactorNumerator',16#10023,pAxisParamters^.fEncScaleFactorNumerator);//fEncScaleFactorNumerator    : LREAL;          (* 0x00010023 *)
_M_MapJsonValues(stAxisMappingJson.stAxisMappingJson[F_Add1(x)],'fEncScaleFactorDenominator',16#10024,pAxisParamters^.fEncScaleFactorDenominator);//fEncScaleFactorDenominator  : LREAL;          (* 0x00010024 *)
//_M_MapJsonValues(stAxisMappingJson[F_Add1(x)],'fEncScaleFactorInternal',16#10024,pAxisParamters^.fEncScaleFactorInternal);//fEncScaleFactorDenominator  : LREAL;          (* 0x00010024 *)
_M_MapJsonValues(stAxisMappingJson.stAxisMappingJson[F_Add1(x)],'fEncOffset',16#10007,pAxisParamters^.fEncOffset);//fEncOffset                  : LREAL;      (* 0x00010007 *)
_M_MapJsonValues(stAxisMappingJson.stAxisMappingJson[F_Add1(x)],'bEncIsInverse',16#10008,pAxisParamters^.bEncIsInverse);//bEncIsInverse               : WORD;       (* 0x00010008 *)
_M_MapJsonValues(stAxisMappingJson.stAxisMappingJson[F_Add1(x)],'fEncModuloFactor',16#10009,pAxisParamters^.fEncModuloFactor);//fEncModuloFactor            : LREAL;      (* 0x00010009 *)
_M_MapJsonValues(stAxisMappingJson.stAxisMappingJson[F_Add1(x)],'nEncMode',16#1000A,pAxisParamters^.nEncMode);//nEncMode                    : DWORD;      (* 0x0001000A *)
_M_MapJsonValues(stAxisMappingJson.stAxisMappingJson[F_Add1(x)],'bEncEnableSoftEndMinControl',16#1000B,pAxisParamters^.bEncEnableSoftEndMinControl);//bEncEnableSoftEndMinControl : WORD;       (* 0x0001000B *)
_M_MapJsonValues(stAxisMappingJson.stAxisMappingJson[F_Add1(x)],'bEncEnableSoftEndMaxControl',16#1000C,pAxisParamters^.bEncEnableSoftEndMaxControl);//bEncEnableSoftEndMaxControl : WORD;       (* 0x0001000C *)
_M_MapJsonValues(stAxisMappingJson.stAxisMappingJson[F_Add1(x)],'fEncSoftEndMin',16#1000D,pAxisParamters^.fEncSoftEndMin);//fEncSoftEndMin              : LREAL;      (* 0x0001000D *)
_M_MapJsonValues(stAxisMappingJson.stAxisMappingJson[F_Add1(x)],'fEncSoftEndMax',16#1000E,pAxisParamters^.fEncSoftEndMax);//fEncSoftEndMax              : LREAL;      (* 0x0001000E *)
_M_MapJsonValues(stAxisMappingJson.stAxisMappingJson[F_Add1(x)],'nEncMaxIncrement',16#10015,pAxisParamters^.nEncMaxIncrement);//nEncMaxIncrement            : DWORD;      (* 0x00010015 *)
_M_MapJsonValues(stAxisMappingJson.stAxisMappingJson[F_Add1(x)],'bEncEnablePosCorrection',16#10016,pAxisParamters^.bEncEnablePosCorrection);//bEncEnablePosCorrection     : WORD;       (* 0x00010016 *)
_M_MapJsonValues(stAxisMappingJson.stAxisMappingJson[F_Add1(x)],'fEncPosCorrectionFilterTime',16#10017,pAxisParamters^.fEncPosCorrectionFilterTime);//fEncPosCorrectionFilterTime : LREAL;      (* 0x00010017 *)
//_M_MapJsonValues(stAxisMappingJson[F_Add1(x)],'nEncReferenceSystem',16#100019,pAxisParamters^.nEncReferenceSystem);//nEncReferenceSystem         : DWORD;          (* 0x00010019 *)
(* CONTROLLER: *)
_M_MapJsonValues(stAxisMappingJson.stAxisMappingJson[F_Add1(x)],'nCtrlId',16#20001,pAxisParamters^.nCtrlId);//nCtrlId                     : DWORD;      (* 0x00020001 *)
_M_MapJsonValues(stAxisMappingJson.stAxisMappingJson[F_Add1(x)],'sCtrlName',16#20002,pAxisParamters^.sCtrlName);//sCtrlName                   : STRING(31); (* 0x00020002 *)
_M_MapJsonValues(stAxisMappingJson.stAxisMappingJson[F_Add1(x)],'nCtrlType',16#20003,pAxisParamters^.nCtrlType);//nCtrlType                   : DWORD;      (* 0x00020003 *)
_M_MapJsonValues(stAxisMappingJson.stAxisMappingJson[F_Add1(x)],'bCtrlEnablePosDiffControl',16#20010,pAxisParamters^.bCtrlEnablePosDiffControl);//bCtrlEnablePosDiffControl   : WORD;       (* 0x00020010 *)
_M_MapJsonValues(stAxisMappingJson.stAxisMappingJson[F_Add1(x)],'bCtrlEnableVeloDiffControl',16#20011,pAxisParamters^.bCtrlEnableVeloDiffControl);//bCtrlEnableVeloDiffControl  : WORD;       (* 0x00020011 *)
_M_MapJsonValues(stAxisMappingJson.stAxisMappingJson[F_Add1(x)],'fCtrlPosDiffMax',16#20012,pAxisParamters^.fCtrlPosDiffMax);//fCtrlPosDiffMax             : LREAL;      (* 0x00020012 *)
_M_MapJsonValues(stAxisMappingJson.stAxisMappingJson[F_Add1(x)],'fCtrlPosDiffMaxTime',16#20012,pAxisParamters^.fCtrlPosDiffMaxTime);//fCtrlPosDiffMaxTime         : LREAL;      (* 0x00020013 *)
_M_MapJsonValues(stAxisMappingJson.stAxisMappingJson[F_Add1(x)],'fCtrlPosKp',16#20102,pAxisParamters^.fCtrlPosKp);//fCtrlPosKp                  : LREAL;      (* 0x00020102 *)
_M_MapJsonValues(stAxisMappingJson.stAxisMappingJson[F_Add1(x)],'fCtrlPosTn',16#20103,pAxisParamters^.fCtrlPosTn);//fCtrlPosTn                  : LREAL;      (* 0x00020103 *)
_M_MapJsonValues(stAxisMappingJson.stAxisMappingJson[F_Add1(x)],'fCtrlPosTv',16#20104,pAxisParamters^.fCtrlPosTv);//fCtrlPosTv                  : LREAL;      (* 0x00020104 *)
_M_MapJsonValues(stAxisMappingJson.stAxisMappingJson[F_Add1(x)],'fCtrlPosTd',16#20105,pAxisParamters^.fCtrlPosTd);//fCtrlPosTd                  : LREAL;      (* 0x00020105 *)
_M_MapJsonValues(stAxisMappingJson.stAxisMappingJson[F_Add1(x)],'fCtrlPosExtKp',16#20106,pAxisParamters^.fCtrlPosExtKp);//fCtrlPosExtKp               : LREAL;      (* 0x00020106 *)
_M_MapJsonValues(stAxisMappingJson.stAxisMappingJson[F_Add1(x)],'fCtrlPosExtVelo',16#20107,pAxisParamters^.fCtrlPosExtVelo);//fCtrlPosExtVelo             : LREAL;      (* 0x00020107 *)
_M_MapJsonValues(stAxisMappingJson.stAxisMappingJson[F_Add1(x)],'fCtrlAccKa',16#20108,pAxisParamters^.fCtrlAccKa);//fCtrlAccKa                  : LREAL;      (* 0x00020108 *)
(* DRIVE: *)
_M_MapJsonValues(stAxisMappingJson.stAxisMappingJson[F_Add1(x)],'nDriveId',16#30001,pAxisParamters^.nDriveId);//nDriveId                    : DWORD;      (* 0x00030001 *)
_M_MapJsonValues(stAxisMappingJson.stAxisMappingJson[F_Add1(x)],'sDriveName',16#30002,pAxisParamters^.sDriveName);//sDriveName                  : STRING(31); (* 0x00030002 *)
_M_MapJsonValues(stAxisMappingJson.stAxisMappingJson[F_Add1(x)],'nDriveType',16#30003,pAxisParamters^.nDriveType);//nDriveType                  : DWORD;      (* 0x00030003 *)
_M_MapJsonValues(stAxisMappingJson.stAxisMappingJson[F_Add1(x)],'bDriveIsInverse',16#30006,pAxisParamters^.bDriveIsInverse);//bDriveIsInverse             : WORD;       (* 0x00030006 *)
_M_MapJsonValues(stAxisMappingJson.stAxisMappingJson[F_Add1(x)],'fDriveVeloReferenz',16#30101,pAxisParamters^.fDriveVeloReferenz);//fDriveVeloReferenz          : LREAL;      (* 0x00030101 *)
_M_MapJsonValues(stAxisMappingJson.stAxisMappingJson[F_Add1(x)],'fDriveOutputReferenz',16#30102,pAxisParamters^.fDriveOutputReferenz);//fDriveOutputReferenz        : LREAL;      (* 0x00030102 *)
_M_MapJsonValues(stAxisMappingJson.stAxisMappingJson[F_Add1(x)],'fDriveOutputScalingAcc',16#3010A,pAxisParamters^.fDriveOutputScalingAcc);//fDriveOutputScalingAcc      : LREAL;        (* 0x0003000A *)
_M_MapJsonValues(stAxisMappingJson.stAxisMappingJson[F_Add1(x)],'fDriveOutputScalingTorque',16#3010C,pAxisParamters^.fDriveOutputScalingTorque);//fDriveOutputScalingTorque   : LREAL;        (* 0x0003000B *)
_M_MapJsonValues(stAxisMappingJson.stAxisMappingJson[F_Add1(x)],'fDriveInputScalingTorque',16#30031,pAxisParamters^.fDriveInputScalingTorque);//fDriveInputScalingTorque    : LREAL;        (* 0x00030031 *)
_M_MapJsonValues(stAxisMappingJson.stAxisMappingJson[F_Add1(x)],'fDriveInputFiltertimeTorque',16#30032,pAxisParamters^.fDriveInputFiltertimeTorque);//fDriveInputFiltertimeTorque : LREAL;        (* 0x00030032 *)
_M_MapJsonValues(stAxisMappingJson.stAxisMappingJson[F_Add1(x)],'fDriveInputFiltertimeTorqueDerivative',16#30033,pAxisParamters^.fDriveInputFiltertimeTorqueDerivative);//fDriveInputFiltertimeTorqueDerivative: LREAL;(* 0x00030033 *)
(* miscellaneous *)
//_M_MapJsonValues(stAxisMappingJson[F_Add1(x)],'fAxisCycleTime',16#00000004,pAxisParamters^.fAxisCycleTime);//fAxisCycleTime              : LREAL;      (* 0x00000004 *) (* available from Tc 2.11 R2 *)
(* 17.05.11: parameter extension *)
_M_MapJsonValues(stAxisMappingJson.stAxisMappingJson[F_Add1(x)],'fRefVeloSearch',16#00000006,pAxisParamters^.fRefVeloSearch);//fRefVeloSearch              : LREAL;      (* 0x00000006 calibration velo (TO plc cam) *)
_M_MapJsonValues(stAxisMappingJson.stAxisMappingJson[F_Add1(x)],'fRefVeloSync',16#00000007,pAxisParamters^.fRefVeloSync);// fRefVeloSync                : LREAL;      (* 0x00000007 calibration velo (off plc cam) *)
_M_MapJsonValues(stAxisMappingJson.stAxisMappingJson[F_Add1(x)],'fVeloSlowManual',16#00000008,pAxisParamters^.fVeloSlowManual);//fVeloSlowManual             : LREAL;      (* 0x00000008 manual velocity (slow) *)
_M_MapJsonValues(stAxisMappingJson.stAxisMappingJson[F_Add1(x)],'fVeloFastManual',16#00000009,pAxisParamters^.fVeloFastManual);//fVeloFastManual             : LREAL;      (* 0x00000009 manual velocity (fast) *)
(* ENCODER (incremental): *)
//_M_MapJsonValues(stAxisMappingJson[F_Add1(x)],'bEncRefSearchInverse',16#10101,pAxisParamters^.bEncRefSearchInverse);//bEncRefSearchInverse        : UINT;       (* 0x00010101 *)
//_M_MapJsonValues(stAxisMappingJson[F_Add1(x)],'bEncRefSyncInverse',16#10102,pAxisParamters^.bEncRefSyncInverse);//bEncRefSyncInverse          : UINT;       (* 0x00010102 *)
//_M_MapJsonValues(stAxisMappingJson[F_Add1(x)],'nEncRefMode',16#10107,pAxisParamters^.nEncRefMode);//nEncRefMode                 : UDINT;      (* 0x00010107 *)
//_M_MapJsonValues(stAxisMappingJson[F_Add1(x)],'fEncRefPosition',16#00010103,pAxisParamters^.fEncRefPosition);//fEncRefPosition             : LREAL;      (* 0x00010103 *)
END_METHOD

METHOD PUBLIC  M_PraseSchemaJson : BOOL
VAR_INPUT
END_VAR
VAR
END_VAR
jsonRoot := THIS^.GetDocumentRoot();
IF jsonRoot > 0 THEN
	M_PraseJsonSchema(jsonRoot,P_sJsonid);
	//M_SetJsonSchema(P_sJsonid.jsonValue,P_sJsonRecipe);
	M_PraseJsonSchema(jsonRoot,P_sJsonValues);
	M_PraseJsonSchema(jsonRoot,P_sJsonTimeStamp);
END_IF
END_METHOD

METHOD PUBLIC M_SetAxisJson : HResult
VAR_INPUT
	lastResult : HRESULT;
	jsonRoot : sJsonValue;
END_VAR
VAR_INPUT
	pAxisParamters : POINTER TO Tc2_MC2.ST_AxisParameterSet;
END_VAR

VAR
	pJson : SJsonValue;
END_VAR

VAR_INST
	saveFile : BOOL;		
	x : UDINT;
	aStringJson : STRING(10000);
	fileName : STRING(255);
	_state			: DINT;
	_fbResult		: FB_ResultHelper;	
	errorCode : HRESULT;
END_VAR
IF _fbResult.M_MethodResult(M_SetAxisJson,lastResult) = FALSE THEN
	RETURN;
ELSE

	IF _fbResult.P_Result = E_Result.S_OK THEN //Reset
		_state := 0;	
		x := 0;
	END_IF 

	_fbResult.P_Result := E_Result.S_WORKING; //Working	
	
	CASE _state OF
		0:
			FOR x := 0 TO NUM_OF_VARS BY 1 DO
				pJson := THIS^.M_SetJsonMember(jsonRoot,stAxisMappingJson.stAxisMappingJson[x].name);		(* 3 Inches *)			
				THIS^.M_SetAxisJson_Values(pJson,ADR(stAxisMappingJson.stAxisMappingJson[x]),(pAxisParamters));
			END_FOR
			_fbResult.P_Result := E_Result.S_OK;
	END_CASE		
END_IF
END_METHOD

METHOD PROTECTED M_SetAxisJson_Values : HResult
VAR_INPUT
	sJson : SJsonValue;
	stAxisMapping : POINTER TO ST_AxisMapping;
	pAxisParamters : POINTER TO Tc2_MC2.ST_AxisParameterSet;
END_VAR
VAR
	pAny : MPM_JsonParser.ST_AnyType_User;	
END_VAR
pAny := stAxisMapping^.pAny; //copy so can be modified 
pAny.pvalue := pAny.pvalue + pAxisParamters; //very important how this works
THIS^.M_SetJsonMemberValue_AnyType(sJson,'value',pAny);
THIS^.M_SetJsonMemberValue(sJson,'indexOffset',stAxisMapping^.indexOffset);
END_METHOD

METHOD PUBLIC M_SetParametersToAxis : HRESULT
VAR_INPUT
	lastResult : HRESULT;
	axisID : DINT;
	pAxisParamters : POINTER TO Tc2_Mc2.ST_AxisParameterSet;
END_VAR
VAR_INST
	adsWrite : ADSWRITE;	
	_state			: DINT;
	_fbResult		: FB_ResultHelper;
	x : DINT;
END_VAR
IF _fbResult.M_MethodResult(M_SetParametersToAxis,lastResult) = FALSE THEN
	RETURN;
ELSE

	IF _fbResult.P_Result = E_Result.S_OK THEN //Reset
		_state := 0;	
		adsWrite(WRITE := FALSE);
		x := 0;
	END_IF 
		
	_fbResult.P_Result := E_Result.S_WORKING; //Working	
	
	CASE _state OF
		0:
			adsWrite.port := PORT;
			adsWrite.IDXGRP := INDEX_BASE + axisID;
			adsWrite.IDXOFFS :=stAxisMappingJson[x].indexOffset;
			adsWrite.LEN := (stAxisMappingJson[x].pAny.diSize);
			adsWrite.SRCADDR := (stAxisMappingJson[x].pAny.pvalue + pAxisParamters);
			adsWrite(WRITE := TRUE);
			_state := 1;
		1:
			adsWrite(WRITE := TRUE);
			IF adsWrite.WRITE = TRUE AND adsWrite.BUSY = FALSE AND adsWrite.ERR = FALSE THEN
				IF x < NUM_OF_VARS THEN
					x := x + 1;
					adsWrite(WRITE := FALSE);
					_state := 0;
				ELSIF x >= NUM_OF_VARS THEN
					_fbResult.P_Result := E_Result.S_OK;
				END_IF
			ELSIF adsWrite.WRITE = TRUE AND adsWrite.BUSY = FALSE AND adsWrite.ERR = TRUE THEN
				ADSLOGSTR(msgCtrlMask := ADSLOG_MSGTYPE_ERROR,
					msgFmtStr := 'Error in %s',
					strArg := stAxisMappingJson[x].name);
				ADSLOGSTR(msgCtrlMask := ADSLOG_MSGTYPE_ERROR,
					msgFmtStr := 'ErrorID %s',
					strArg := TO_STRING(adsWrite.ERRID));
				IF x < NUM_OF_VARS THEN
					x := x + 1;
					adsWrite(WRITE := FALSE);
					_state := 0;
				ELSIF x >= NUM_OF_VARS THEN
					_fbResult.P_Result := E_Result.S_OK;
				END_IF
			END_IF	
	END_CASE
	
END_IF
END_METHOD

END_FUNCTION_BLOCK

// ---- FUN/F_Add1.TcPOU
FUNCTION F_Add1 : DINT
VAR_INPUT
	x : REFERENCE TO DINT;
END_VAR

F_Add1.F_Add1 := x;
x := x + 1;

END_FUNCTION

// ---- FBs/Main/FB_Pump.TcPOU
FUNCTION_BLOCK FB_Pump EXTENDS FB_ConfigBase
VAR_INPUT
END_VAR
VAR_OUTPUT
	fbEventEnable : FB_DiscreteEvents(THIS,3,0,0);	
	fbEventHomePump : FB_DiscreteEvents(THIS,4,0,0);	
	fbEventMoveAbs : FB_DiscreteEvents(THIS,5,ADR(mcMoveAbs),SIZEOF(mcMoveAbs));	
	fbEventMoveHalt : FB_DiscreteEvents(THIS,6,0,0);			
	fbEventPumpContinuous : FB_DiscreteEvents(THIS,7,0,0);			
	fbEventPumpInterminate : FB_DiscreteEvents(THIS,8,0,0);		
END_VAR
VAR
	axis : Tc2_MC2.AXIS_REF;		
	var1 : DINT;
	var2 : STRING;
	ioVar : POINTER TO BOOL;
	ioVar2 : POINTER TO REAL;
	fbAxisControl : FB_AxisControl(axis);
END_VAR

VAR
	testIO : BOOL;
	closeFeedBack : BOOL;
	openFeedBack : BOOL;
END_VAR


VAR
	mcMoveAbs : ARRAY [0..4] OF MPM_JsonParser.ST_AnyType_User := [
	(name := 'Position', typeclass := MPM_JsonParser.E_TypeClassEx.TYPE_LREAL, diSize := SIZEOF(LREAL)),
	(name := 'Velocity', typeclass := MPM_JsonParser.E_TypeClassEx.TYPE_LREAL, diSize := SIZEOF(LREAL)),	
	(name := 'Acceleration', typeclass := MPM_JsonParser.E_TypeClassEx.TYPE_LREAL, diSize := SIZEOF(LREAL)),
	(name := 'Deceleration', typeclass := MPM_JsonParser.E_TypeClassEx.TYPE_LREAL, diSize := SIZEOF(LREAL)),	
	(name := 'Jerk', typeclass := MPM_JsonParser.E_TypeClassEx.TYPE_LREAL, diSize := SIZEOF(LREAL))	
	];		
END_VAR

//axis
VAR
	stAxisParameterSet : Tc2_MC2.ST_AxisParameterSet;  
END_VAR
//IO

VAR
	//Recipe tags
	//Intermient Move
	volume : LREAL := 100; // this will set number of revs
	timeToDispense : LREAL := 10; //time to dispence 
	//Continous mode
	volumePerSecond : LREAL;
	highLevelOverride : LREAL;
	lowLevelOverride : LREAL;
	//System tags
	volumePerRotation : LREAL; //0.23 liters for pump
	//IO
	lowLevelSensor : BOOL;
	HighLevelSensor : BOOL;
	
	fbKinenmatics2 : FB_Kinenmatics_V2;	
END_VAR

METHOD _F_Axis : HRESULT
VAR_IN_OUT
	a_pstAxisParameterSet : POINTER TO Tc2_MC2.ST_AxisParameterSet; //pointer to array
	pstAxisMapping : UDINT;
END_VAR
stAxisParameterSet.AxisId := axis.NcToPlc.AxisId;
a_pstAxisParameterSet := ADR(stAxisParameterSet);
pstAxisMapping := SIZEOF(stAxisParameterSet);

_F_Axis := MPM_FBResult.E_Result.S_OK;
END_METHOD

METHOD PROTECTED  _F_IO : HResult
VAR_IN_OUT
	a_pstIOMappingJson : POINTER TO ST_IOMappingJson; //pointer to array
	ustIOMappingJson : UDINT; 		
END_VAR
VAR_INST
	stIOMappingJson : ARRAY [0..1] OF ST_IOMappingJson;
END_VAR
VAR
	x : DINT;
END_VAR
//	ioVar : POINTER TO BOOL;
//	ioVar2 : POINTER TO REAL;
F_Map_ST_IOMappingJson(ADR(a_pstIOMappingJson[F_Add1(x)]),'lowLevelSensor',ADR(lowLevelSensor));
F_Map_ST_IOMappingJson(ADR(a_pstIOMappingJson[F_Add1(x)]),'HighLevelSensor',ADR(HighLevelSensor));

a_pstIOMappingJson := ADR(stIOMappingJson);
ustIOMappingJson := SIZEOF(stIOMappingJson);




_F_IO := MPM_FBResult.E_Result.S_OK;
END_METHOD

(*
return the list of vars that want to be saved and loaded 
*)

METHOD PROTECTED  _F_Recipe : HResult
VAR_IN_OUT
	a_pstAnyTypeUser : POINTER TO MPM_JsonParser.ST_AnyType_User; //pointer to array
	uAnyTypeUser : UDINT; //size of array	
END_VAR
VAR_OUTPUT
END_VAR
VAR
	x : DINT;
END_VAR
VAR_INST
	a_stAnyTypeUser : ARRAY [0..1] OF MPM_JsonParser.ST_AnyType_User;
END_VAR
MPM_JsonParser.F_Map_ST_AnyType_User('volume',volume,a_stAnyTypeUser[F_Add1(x)]);
MPM_JsonParser.F_Map_ST_AnyType_User('timeToDispense',timeToDispense,a_stAnyTypeUser[F_Add1(x)]);


a_pstAnyTypeUser := ADR(a_stAnyTypeUser);
uAnyTypeUser := SIZEOF(a_stAnyTypeUser);

_F_Recipe := MPM_FBResult.E_Result.S_OK;
END_METHOD

METHOD PROTECTED _F_System : HResult
VAR_IN_OUT
	a_pstAnyTypeUser : POINTER TO MPM_JsonParser.ST_AnyType_User; //pointer to array
	uAnyTypeUser : UDINT; //size of array	
END_VAR
VAR_INST
	a_stAnyTypeUser : ARRAY [0..0] OF MPM_JsonParser.ST_AnyType_User;
END_VAR
VAR
	x : DINT;
END_VAR
MPM_JsonParser.F_Map_ST_AnyType_User('volumePerRotation',volumePerRotation,a_stAnyTypeUser[F_Add1(x)]);


a_pstAnyTypeUser := ADR(a_stAnyTypeUser);
uAnyTypeUser := SIZEOF(a_stAnyTypeUser);

_F_System := MPM_FBResult.E_Result.S_OK;
END_METHOD

METHOD FB_init : BOOL
VAR_INPUT
	bInitRetains : BOOL; // if TRUE, the retain variables are initialized (warm start / cold start)
	bInCopyCode : BOOL;  // if TRUE, the instance afterwards gets moved into the copy code (online change)
	fbName : STRING;
END_VAR
END_METHOD

METHOD PROTECTED M_CloseValve : HResult
VAR_INPUT
	lastResult : HResult;	
END_VAR
VAR_INST
	_lastResult : HResult;
	_fbResult : FB_ResultHelper_V2_1;
	_state : DINT;
END_VAR
IF _fbResult.M_MethodResult(M_CloseValve,lastResult,ADR(_lastResult)) = FALSE THEN
	RETURN;
END_IF

IF _fbResult.P_MethodResult = E_Result.S_OK THEN
	_state := 0;
END_IF


_fbResult.P_MethodResult := E_Result.S_WORKING;


CASE _state OF 
	0:
		testIO := TRUE;
		IF closeFeedBack = TRUE THEN
			_fbResult.P_MethodResult := E_Result.S_OK;
		END_IF
END_CASE
END_METHOD

METHOD PUBLIC  M_Events : HResult
VAR_INPUT
	lastResult : HResult;
	eventID : DINT;
END_VAR
VAR_INST
	_fbResult : FB_ResultHelper_V2_1;
	_lastResult : HResult;
	openValve_Result : HRESULT;
	closeValve_Result : HRESULT;
	enablePump_Result : HRESULT;
	homeDirect_Result : HRESULT; 
	moveABS_Result : HRESULT; 	
	moveInter_Result : HRESULT; 		
	moveVelocity_Result : HRESULT; 		
	halt_Result : HRESULT;
END_VAR
VAR 
	HomingMode : Tc2_MC2.MC_HomingMode;
	OptionsHomeing : Tc2_MC2.ST_HomingOptions;
	BufferMode : Tc2_MC2.MC_BufferMode;
	OptionsPower : Tc2_MC2.ST_PowerOptions;	
	Options : Tc2_MC2.ST_MoveOptions;		
END_VAR

VAR_INST
	executeDyn : BOOL;
	VelocityDyn : LREAL := 10; 
END_VAR
CASE eventID OF 
	1 : //Open Valve
		IF _fbResult.M_MethodResult(M_Events,lastResult,ADR(openValve_Result)) = FALSE THEN
			RETURN;
		END_IF
		IF closeValve_Result > E_Result.S_OK THEN
			closeValve_Result := -1; //fail it out
		END_IF	
		_fbResult.P_MethodResult := M_OpenValve(_fbResult.P_MethodResult);
	2:
		IF _fbResult.M_MethodResult(M_Events,lastResult,ADR(closeValve_Result)) = FALSE THEN
			RETURN;
		END_IF
		IF openValve_Result > E_Result.S_OK THEN
			openValve_Result := -1; //fail it out
		END_IF
		_fbResult.P_MethodResult := M_CloseValve(_fbResult.P_MethodResult);	
	3: //enable pump
		IF _fbResult.M_MethodResult(M_Events,lastResult,ADR(enablePump_Result)) = FALSE THEN
			RETURN;
		END_IF	
		_fbResult.P_MethodResult := fbAxisControl.MC_Power(_fbResult.P_MethodResult,TRUE,TRUE,TRUE,100.0,BufferMode,OptionsPower);
	4: //Home Pump
		IF _fbResult.M_MethodResult(M_Events,lastResult,ADR(homeDirect_Result)) = FALSE THEN
			RETURN;
		END_IF			
		HomingMode := Tc2_MC2.MC_HomingMode.MC_Direct; 
		_fbResult.P_MethodResult := fbAxisControl.MC_Home(_fbResult.P_MethodResult,0.0,HomingMode,BufferMode,OptionsHomeing);
	5: //move pump absoulte
		IF _fbResult.M_MethodResult(M_Events,lastResult,ADR(moveABS_Result)) = FALSE THEN
			RETURN;
		END_IF		
		_fbResult.P_MethodResult := fbAxisControl.MC_MoveAbsoulte(_fbResult.P_MethodResult,
			Position := F_TO_LREAL(mcMoveAbs[0].pvalue),
			Velocity := F_TO_LREAL(mcMoveAbs[1].pvalue),
			Acceleration := F_TO_LREAL(mcMoveAbs[2].pvalue),
			Deceleration := F_TO_LREAL(mcMoveAbs[3].pvalue),
			Jerk := F_TO_LREAL(mcMoveAbs[4].pvalue),
			BufferMode := BufferMode,
			Options := Options);	
	6: //halt pump
		IF _fbResult.M_MethodResult(M_Events,lastResult,ADR(halt_Result)) = FALSE THEN
			RETURN;
		END_IF			
		_fbResult.P_MethodResult := fbAxisControl.MC_Halt(_fbResult.P_MethodResult,
			1000.0,
			1000.0);				
	7: //pump_continuous
	IF _fbResult.M_MethodResult(M_Events,lastResult,ADR(moveVelocity_Result)) = FALSE THEN
			RETURN;
		END_IF		
		VelocityDyn := VelocityDyn + 0.10;
		IF VelocityDyn > 1000 THEN
			VelocityDyn := 10;
		END_IF
		_fbResult.P_MethodResult := fbAxisControl.MC_MoveVelocityDyn(
			_fbResult.P_MethodResult,
			Direction := Tc2_MC2.MC_Direction.MC_Positive_Direction,
			executeDyn,
			VelocityDyn,			
			1000,
			1000,
			10000,
			BufferMode,
			Options);	
	8: //pump_intermeate
	fbKinenmatics2.jerkLimit := 100000;
	fbKinenmatics2.accelLimit := 15000.0;	
	fbKinenmatics2.decelLimit := 15000.0;	
	fbKinenmatics2.velocityLimit := 2500;	
	fbKinenmatics2.positionDelta := volume;		
	fbKinenmatics2.timeToComplete := timeToDispense;
	fbKinenmatics2();
	IF _fbResult.M_MethodResult(M_Events,lastResult,ADR(moveInter_Result)) = FALSE THEN
			RETURN;
		END_IF		
		_fbResult.P_MethodResult := fbAxisControl.MC_MoveRelative(
			_fbResult.P_MethodResult,
			volume,
			fbKinenmatics2.velocityOutput,
			fbKinenmatics2.accelOutput,			
			fbKinenmatics2.decelLimit,		
			fbKinenmatics2.jerkOutput,		
			BufferMode,
			Options);			
END_CASE
END_METHOD

METHOD PUBLIC M_Execute : HRESULT
VAR_INPUT
END_VAR
fbAxisControl.M_Execute();
END_METHOD

METHOD M_GetEvent : HResult
VAR_INPUT
	pFbDiscreteEvents : POINTER TO POINTER TO FB_DiscreteEvents;
	index : DINT;
END_VAR
CASE index OF
	0:
		pFbDiscreteEvents^ := ADR(fbEventEnable);
	1:
		pFbDiscreteEvents^ := ADR(fbEventHomePump);	
	2:
		pFbDiscreteEvents^ := ADR(fbEventMoveAbs);
	3:
		pFbDiscreteEvents^ := ADR(fbEventMoveHalt);	
	4:
		pFbDiscreteEvents^ := ADR(fbEventPumpContinuous);	
	5:
		pFbDiscreteEvents^ := ADR(fbEventPumpInterminate);	
	ELSE
		M_GetEvent := E_Result.S_FAILED;								
END_CASE
END_METHOD

{attribute 'TcRpcEnable'}
METHOD PUBLIC M_HMI_SET_VOLUME : HRESULT
VAR_INPUT
	value : LREAL;
END_VAR
VAR_OUTPUT
	errorMsg : STRING(256);
END_VAR
IF value < 0 THEN
	M_HMI_SET_VOLUME := E_Result.S_FAILED;
	errorMsg := 'value cant be less than 0';
	RETURN;
ELSE
	volume := value;
END_IF
END_METHOD

METHOD PROTECTED M_OpenValve : HResult
VAR_INPUT
	lastResult : HResult;	
END_VAR
VAR_INST
	_lastResult : HResult;
	_fbResult : FB_ResultHelper_V2_1;
	_state : DINT;	
END_VAR
IF _fbResult.M_MethodResult(M_OpenValve,lastResult,ADR(_lastResult)) = FALSE THEN
	RETURN;
END_IF

IF _fbResult.P_MethodResult = E_Result.S_OK THEN
	_state := 0;
END_IF


_fbResult.P_MethodResult := E_Result.S_WORKING;


CASE _state OF 
	0:
		testIO := FALSE;
		IF openFeedBack = TRUE THEN
			_fbResult.P_MethodResult := E_Result.S_OK;
		END_IF
END_CASE
END_METHOD

PROPERTY P_GetNumOfEvents : DINT
GET
P_GetNumOfEvents := 6; //0..5
END_GET
END_PROPERTY

END_FUNCTION_BLOCK

// ---- FBs/Abstracts/FB_AxisControl.TcPOU
(*
Standard control for FB_AxisRef
*)

FUNCTION_BLOCK FB_AxisControl
VAR_INPUT
	
END_VAR
VAR_OUTPUT
END_VAR
VAR
	axisRef : REFERENCE TO Tc2_MC2.AXIS_REF;	
	fbMCPower : Tc2_MC2.MC_Power;
	fbMCReset : Tc2_MC2.MC_Reset;		
	fbMCHome : Tc2_MC2.MC_Home;
	fbMCStop : Tc2_MC2.MC_Stop;
	fbMCHalt :  Tc2_MC2.MC_Halt;
	axisState : Tc2_MC2.MC_AxisStates;
	
	//Discrete motion
	fbMCMoveAbsolute : Tc2_MC2.MC_MoveAbsolute;
	fbMCMoveRelative : Tc2_MC2.MC_MoveRelative;
	fbMoveVelocity : Tc2_MC2.MC_MoveVelocity;
	fbMoveVelocityDyn : ARRAY [0..1] OF Tc2_MC2.MC_MoveVelocity;
	//Axis Coupling
	fbGearInDyn : Tc2_MC2.MC_GearInDyn;
	fbGearOut : Tc2_MC2.MC_GearOut;
	
	//Phasing
	fbPhasingAbsolute : Tc2_MC2.MC_PhasingAbsolute;
	fbHaltPhasing : Tc2_MC2.MC_HaltPhasing;
	fbPhasingRelative: Tc2_MC2.MC_PhasingRelative;
	
END_VAR

METHOD FB_init : BOOL
VAR_INPUT
	bInitRetains : BOOL; // if TRUE, the retain variables are initialized (warm start / cold start)
	bInCopyCode : BOOL;  // if TRUE, the instance afterwards gets moved into the copy code (online change)
	axisRef : REFERENCE TO Tc2_MC2.AXIS_REF;		
END_VAR
THis^.axisRef rEF= axisRef;
END_METHOD

METHOD M_Execute : BOOL
VAR_INPUT
END_VAR
axisRef.ReadStatus();
END_METHOD

METHOD MC_Halt : HResult
VAR_INPUT
	lastResult : HResult;
	Deceleration : LREAL; 
	Jerk : LREAL;
END_VAR
VAR_OUTPUT
	Busy : BOOL;
	Active : BOOL;
	Error : BOOL;
	ErrorID : UDINT;	
END_VAR
VAR_INST
	_fbResult : FB_ResultHelper_V2_1;
	_lastResult : HResult;	
	_state : DINT;
END_VAR
IF _fbResult.M_MethodResult(MC_Halt,lastResult,ADR(_lastResult)) = FALSE THEN
	RETURN;
END_IF

IF _fbResult.P_MethodResult = E_Result.S_OK THEN
	_state := 0;
	fbMCHalt(Axis := axisRef, Execute  := FALSE,Deceleration := Deceleration,Jerk := Jerk);	
END_IF


_fbResult.P_MethodResult := E_Result.S_WORKING;

CASE _state OF
	0:
		fbMCHalt(Axis := axisRef, Execute  := TRUE,Deceleration := Deceleration,Jerk := Jerk);
		_state := 1;
	1:
		fbMCHalt(Axis := axisRef,Execute  := TRUE);	
		IF fbMCHalt.Done = TRUE AND fbMCHalt.Error = FALSE THEN
			_fbResult.P_MethodResult := E_Result.S_OK;
		ELSIF fbMCHalt.Done = FALSE AND fbMCHalt.Error = TRUE THEN 
			_fbResult.P_MethodResult := E_Result.S_FAILED;
		ELSIF fbMCHalt.CommandAborted = TRUE AND fbMCHalt.Error = FALSE THEN 
			_fbResult.P_MethodResult := E_Result.S_FAILED;			
		END_IF		
END_CASE
END_METHOD

METHOD PUBLIC MC_Home : HResult
VAR_INPUT
	lastResult : HResult;
	Position : LREAL;	
	HomingMode : Tc2_MC2.MC_HomingMode;
	BufferMode : Tc2_MC2.MC_BufferMode;
	Options : Tc2_MC2.ST_HomingOptions;
END_VAR
VAR_OUTPUT
	Done : BOOL;
	Busy : BOOL;
	Active : BOOL;
	CommandAborted : BOOL;
	Error : BOOL;
	ErrorID : UDINT;		
END_VAR
VAR_INST
	_fbResult : FB_ResultHelper_V2_1;
	_lastResult : HResult;	
	_state : DINT;
END_VAR
IF _fbResult.M_MethodResult(MC_Home,lastResult,ADR(_lastResult)) = FALSE THEN
	RETURN;
END_IF

IF _fbResult.P_MethodResult = E_Result.S_OK THEN
	_state := 0;
	fbMCHome(axis := axisRef,Execute := FALSE);
END_IF


_fbResult.P_MethodResult := E_Result.S_WORKING;

CASE _state OF
	0:
		fbMCHome(Axis := axisRef,
			Execute := TRUE,
			Position := Position,
			HomingMode := HomingMode,
			BufferMode := BufferMode,
			Options := Options,
			Done => Done, 
			Busy => Busy, 
			Active => Active, 
			CommandAborted => CommandAborted, 
			Error => Error, 
			ErrorID => ErrorID);
		_state := 1;
	1:
		fbMCHome(Axis := axisRef,			
			Done => Done, 
			Busy => Busy, 
			Active => Active, 
			CommandAborted => CommandAborted, 
			Error => Error, 
			ErrorID => ErrorID);	
		IF fbMCHome.Done = TRUE AND fbMCHome.Error = FALSE THEN
			_fbResult.P_MethodResult := E_Result.S_OK;
		ELSIF fbMCHome.Done = TRUE AND fbMCHome.Error = TRUE THEN 
			_fbResult.P_MethodResult := E_Result.S_FAILED;
		ELSIF fbMCHalt.CommandAborted = TRUE AND fbMCHalt.Error = FALSE THEN 
			_fbResult.P_MethodResult := E_Result.S_FAILED;						
		END_IF		
END_CASE
END_METHOD

METHOD PUBLIC MC_MoveAbsoulte : HResult
VAR_INPUT
	lastResult : HResult;
	Position : LREAL;	
	Velocity : LREAL;
	Acceleration : LREAL;
	Deceleration : LREAL;
	Jerk : LREAL;
	BufferMode : Tc2_MC2.MC_BufferMode;
	Options : Tc2_MC2.ST_MoveOptions;	
END_VAR
VAR_OUTPUT
	Done : BOOL;
	Active : BOOL;
	CommandAborted : BOOL;
	Error : BOOL;
	ErrorID : UDINT;	
END_VAR
VAR_INST
	_fbResult : FB_ResultHelper_V2_1;
	_lastResult : HResult;	
	_state : DINT;
END_VAR
IF _fbResult.M_MethodResult(MC_MoveAbsoulte,lastResult,ADR(_lastResult)) = FALSE THEN
	RETURN;
END_IF

IF _fbResult.P_MethodResult = E_Result.S_OK THEN
	_state := 0;
	fbMCMoveAbsolute(axis := axisRef,Execute := FALSE);
END_IF


_fbResult.P_MethodResult := E_Result.S_WORKING;

CASE _state OF
	0:
		fbMCMoveAbsolute(Axis := axisRef,
			Execute := TRUE,
			Position := Position,
			Velocity := Velocity,
			Acceleration := Acceleration,
			Deceleration := Deceleration,
			Jerk := Jerk,
			BufferMode := BufferMode,
			Options := Options,
			Done => Done,
			Active => Active,
			CommandAborted => CommandAborted,
			Error => Error,
			ErrorID => ErrorID);
		_state := 1;
	1:
		fbMCMoveAbsolute(Axis := axisRef,			
			Done => Done,
			Active => Active,
			CommandAborted => CommandAborted,
			Error => Error,
			ErrorID => ErrorID);	
		IF fbMCMoveAbsolute.Done = TRUE AND fbMCMoveAbsolute.Error = FALSE THEN
			_fbResult.P_MethodResult := E_Result.S_OK;
		ELSIF fbMCMoveAbsolute.Done = TRUE AND fbMCMoveAbsolute.Error = TRUE THEN 
			_fbResult.P_MethodResult := E_Result.S_FAILED;
		ELSIF fbMCMoveAbsolute.CommandAborted = TRUE AND fbMCMoveAbsolute.Error = FALSE THEN 
			_fbResult.P_MethodResult := E_Result.S_FAILED;					
		END_IF		
END_CASE
END_METHOD

METHOD PUBLIC MC_MoveRelative : HResult
VAR_INPUT
	lastResult : HResult;
	Distance : LREAL;	
	Velocity : LREAL;
	Acceleration : LREAL;
	Deceleration : LREAL;
	Jerk : LREAL;
	BufferMode : Tc2_MC2.MC_BufferMode;
	Options : Tc2_MC2.ST_MoveOptions;	
END_VAR
VAR_OUTPUT
	Done : BOOL;
	Active : BOOL;
	CommandAborted : BOOL;
	Error : BOOL;
	ErrorID : UDINT;	
END_VAR
VAR_INST
	_fbResult : FB_ResultHelper_V2_1;
	_lastResult : HResult;	
	_state : DINT;
END_VAR
IF _fbResult.M_MethodResult(MC_MoveRelative,lastResult,ADR(_lastResult)) = FALSE THEN
	RETURN;
END_IF

IF _fbResult.P_MethodResult = E_Result.S_OK THEN
	_state := 0;
	fbMCMoveRelative(axis := axisRef,Execute := FALSE);
END_IF


_fbResult.P_MethodResult := E_Result.S_WORKING;

CASE _state OF
	0:
		fbMCMoveRelative(Axis := axisRef,
			Execute := TRUE,
			Distance := Distance,
			Velocity := Velocity,
			Acceleration := Acceleration,
			Deceleration := Deceleration,
			Jerk := Jerk,
			BufferMode := BufferMode,
			Options := Options,
			Done => Done,
			Active => Active,
			CommandAborted => CommandAborted,
			Error => Error,
			ErrorID => ErrorID);
		_state := 1;
	1:
		fbMCMoveRelative(Axis := axisRef,
			Done => Done,
			Active => Active,
			CommandAborted => CommandAborted,
			Error => Error,
			ErrorID => ErrorID);	
		IF fbMCMoveRelative.Done = TRUE AND fbMCMoveRelative.Error = FALSE THEN
			_fbResult.P_MethodResult := E_Result.S_OK;
		ELSIF fbMCMoveRelative.Done = TRUE AND fbMCMoveRelative.Error = TRUE THEN 
			_fbResult.P_MethodResult := E_Result.S_FAILED;
		ELSIF fbMCMoveRelative.CommandAborted = TRUE AND fbMCMoveRelative.Error = FALSE THEN 
			_fbResult.P_MethodResult := E_Result.S_FAILED;		
		END_IF		
END_CASE
END_METHOD

METHOD PUBLIC MC_MoveVelocity : HResult
VAR_INPUT
	lastResult : HResult;
	Direction : Tc2_MC2.MC_Direction;	
	Velocity : LREAL;
	Acceleration : LREAL;
	Deceleration : LREAL;
	Jerk : LREAL;
	BufferMode : Tc2_MC2.MC_BufferMode;
	Options : Tc2_MC2.ST_MoveOptions;	
END_VAR
VAR_OUTPUT
	InVelocity : BOOL;
	Busy : BOOL;
	Active : BOOL;
	CommandAborted : BOOL;
	Error : BOOL;
	ErrorID : UDINT;	
END_VAR
VAR_INST
	_fbResult : FB_ResultHelper_V2_1;
	_lastResult : HResult;	
	_state : DINT;
END_VAR
IF _fbResult.M_MethodResult(MC_MoveVelocity,lastResult,ADR(_lastResult)) = FALSE THEN
	RETURN;
END_IF

IF _fbResult.P_MethodResult = E_Result.S_OK THEN
	_state := 0;
	fbMoveVelocity(axis := axisRef,Execute := FALSE);
END_IF


_fbResult.P_MethodResult := E_Result.S_WORKING;

CASE _state OF
	0:
		fbMoveVelocity(Axis := axisRef,
			Execute := TRUE,
			Direction := Direction,
			Velocity := Velocity,
			Acceleration := Acceleration,
			Deceleration := Deceleration,
			Jerk := Jerk,
			BufferMode := BufferMode,
			Options := Options,
			InVelocity => InVelocity,
			Busy => Busy,
			Active => Active,
			CommandAborted => CommandAborted,
			Error => Error,
			ErrorID => ErrorID);
		_state := 1;
	1:
		fbMoveVelocity(Axis := axisRef,			
			Busy => Busy,
			Active => Active,
			CommandAborted => CommandAborted,
			Error => Error,
			ErrorID => ErrorID);
		IF fbMoveVelocity.InVelocity = TRUE AND fbMoveVelocity.Error = FALSE THEN
			_fbResult.P_MethodResult := E_Result.S_OK;
		ELSIF fbMoveVelocity.InVelocity = TRUE AND fbMoveVelocity.Error = TRUE THEN 
			_fbResult.P_MethodResult := E_Result.S_FAILED;
		ELSIF fbMoveVelocity.CommandAborted = TRUE AND fbMoveVelocity.Error = FALSE THEN 
			_fbResult.P_MethodResult := E_Result.S_FAILED;					
		END_IF		
END_CASE
END_METHOD

METHOD PUBLIC MC_MoveVelocityDyn : HResult
VAR_INPUT
	lastResult : HResult;
	Direction : Tc2_MC2.MC_Direction;	
	Execute : BOOL;
	Velocity : LREAL;
	Acceleration : LREAL;
	Deceleration : LREAL;
	Jerk : LREAL;
	BufferMode : Tc2_MC2.MC_BufferMode;
	Options : Tc2_MC2.ST_MoveOptions;	
END_VAR
VAR_OUTPUT
	InVelocity : BOOL;
	Busy : BOOL;
	Active : BOOL;
	CommandAborted : BOOL;
	Error : BOOL;
	ErrorID : UDINT;	
END_VAR
VAR_INST
	_Velocity : LREAL;
	_fbResult : FB_ResultHelper_V2_1;
	_lastResult : HResult;	
	_state : DINT;
	fbMoveVelocityDyn : POINTER TO Tc2_MC2.MC_MoveVelocity;	
END_VAR
IF _fbResult.M_MethodResult(MC_MoveVelocityDyn,lastResult,ADR(_lastResult)) = FALSE THEN
	RETURN;
END_IF

IF _fbResult.P_MethodResult = E_Result.S_OK THEN
	_state := 0;
	THIS^.fbMoveVelocityDyn[0](Axis := axisRef ,Execute := FALSE);
	THIS^.fbMoveVelocityDyn[1](Axis := axisRef ,Execute := FALSE);	
END_IF
IF Execute = TRUE THEN
	IF THIS^.fbMoveVelocityDyn[0].Busy = FALSE AND THIS^.fbMoveVelocityDyn[0].Busy = FALSE THEN //if no function is running pick 0
		fbMoveVelocityDyn := ADR(THIS^.fbMoveVelocityDyn[0]);
	ELSIF _Velocity = Velocity AND THIS^.fbMoveVelocityDyn[0].Busy = TRUE THEN //if 
		fbMoveVelocityDyn := ADR(THIS^.fbMoveVelocityDyn[0]);
		THIS^.fbMoveVelocityDyn[1](Axis := axisRef ,Execute := FALSE);	
	ELSIF _Velocity = Velocity AND THIS^.fbMoveVelocityDyn[1].Busy = TRUE THEN
		fbMoveVelocityDyn := ADR(THIS^.fbMoveVelocityDyn[1]);
		THIS^.fbMoveVelocityDyn[0](Axis := axisRef ,Execute := FALSE);
		_state := 0;	
	ELSIF _Velocity <> Velocity AND THIS^.fbMoveVelocityDyn[0].Busy = FALSE THEN
		fbMoveVelocityDyn := ADR(THIS^.fbMoveVelocityDyn[0]);
		THIS^.fbMoveVelocityDyn[1](Axis := axisRef ,Execute := FALSE);
		_state := 0;
	ELSIF _Velocity <> Velocity AND THIS^.fbMoveVelocityDyn[1].Busy = FALSE THEN
		fbMoveVelocityDyn := ADR(THIS^.fbMoveVelocityDyn[1]);
		THIS^.fbMoveVelocityDyn[0](Axis := axisRef ,Execute := FALSE);
		_state := 0;
	ELSE //Something is wrong
		_fbResult.P_MethodResult := E_Result.S_WORKING;
		THIS^.fbMoveVelocityDyn[0](Axis := axisRef ,Execute := FALSE);
		THIS^.fbMoveVelocityDyn[1](Axis := axisRef ,Execute := FALSE);
		RETURN;
	END_IF
	
	_fbResult.P_MethodResult := E_Result.S_WORKING;
	
	
ELSE //execute value is low check to see if any functions are still running if not then return S_OK
	IF THIS^.fbMoveVelocityDyn[0].Busy THEN
		fbMoveVelocityDyn := ADR(THIS^.fbMoveVelocityDyn[0]);
		_fbResult.P_MethodResult := E_Result.S_WORKING;
	ELSIF THIS^.fbMoveVelocityDyn[1].Busy THEN
		fbMoveVelocityDyn := ADR(THIS^.fbMoveVelocityDyn[1]);
		_fbResult.P_MethodResult := E_Result.S_WORKING;
	ELSE
		_fbResult.P_MethodResult := E_Result.S_OK;		
	END_IF
END_IF







CASE _state OF
	0:
		_Velocity := Velocity;
		fbMoveVelocityDyn^(Axis := axisRef,
			Execute := Execute,
			Direction := Direction,
			Velocity := Velocity,
			Acceleration := Acceleration,
			Deceleration := Deceleration,
			Jerk := Jerk,
			BufferMode := BufferMode,
			Options := Options,
			InVelocity => InVelocity,
			Busy => Busy,
			Active => Active,
			CommandAborted => CommandAborted,
			Error => Error,
			ErrorID => ErrorID);
		IF Execute = FALSE AND fbMoveVelocity.InVelocity = TRUE AND fbMoveVelocity.Error = FALSE THEN //Execute has to be false the retrun S_OK
			_fbResult.P_MethodResult := E_Result.S_OK;
		ELSIF Execute = FALSE AND fbMoveVelocity.InVelocity = TRUE AND fbMoveVelocity.Error = TRUE THEN 
			_fbResult.P_MethodResult := E_Result.S_FAILED;
		ELSIF Execute = TRUE AND fbMoveVelocity.Busy = FALSE THEN
			fbMoveVelocityDyn^(Axis := axisRef, Execute := FALSE);
		END_IF		
END_CASE
END_METHOD

METHOD PUBLIC MC_Power : HResult
VAR_INPUT
	lastResult : HResult;
	Enable : BOOL;
	Enable_Negative : BOOL;
	Enable_Positive : BOOL;
	Override : LREAL;
	BufferMode : Tc2_MC2.MC_BufferMode;
	Options : Tc2_MC2.ST_PowerOptions;
END_VAR
VAR_OUTPUT
	Busy : BOOL;
	Active : BOOL;
	Error : BOOL;
	ErrorID : UDINT;	
END_VAR
VAR_INST
	_fbResult : FB_ResultHelper_V2_1;
	_lastResult : HResult;	
	_state : DINT;
END_VAR
IF _fbResult.M_MethodResult(MC_Power,lastResult,ADR(_lastResult)) = FALSE THEN
	RETURN;
END_IF

	fbMCPower(axis := axisRef);

IF _fbResult.P_MethodResult = E_Result.S_OK  AND Enable = TRUE AND fbMCPower.Busy = TRUE THEN //if running allready return S_OK
	_fbResult.P_MethodResult := E_Result.S_WORKING;
	RETURN;
ELSIF _fbResult.P_MethodResult = E_Result.S_OK THEN 	
	_state := 0;
	fbMCPower(axis := axisRef,Enable := FALSE);
END_IF



_fbResult.P_MethodResult := E_Result.S_WORKING;

CASE _state OF
	0:
		fbMCPower(Axis := axisRef, 
			Enable := Enable,
			Enable_Negative := Enable_Negative,
			Enable_Positive := Enable_Positive,
			Override := Override,
			BufferMode := BufferMode, 
			Options := Options, 
			Busy => Busy, 
			Active => Active, 
			Error => Error, 
			ErrorID => ErrorID);
		IF fbMCPower.Busy = FALSE AND fbMCPower.Error = FALSE THEN
			_fbResult.P_MethodResult := E_Result.S_OK;
		ELSIF fbMCPower.Busy = FALSE AND fbMCPower.Error = TRUE THEN 
			_fbResult.P_MethodResult := E_Result.S_FAILED;
		END_IF		
END_CASE
END_METHOD

METHOD PUBLIC MC_Reset : HResult
VAR_INPUT
	lastResult : HResult;
END_VAR
VAR_OUTPUT
	Busy : BOOL;
	Active : BOOL;
	Error : BOOL;
	ErrorID : UDINT;	
END_VAR
VAR_INST
	_fbResult : FB_ResultHelper_V2_1;
	_lastResult : HResult;	
	_state : DINT;
END_VAR
IF _fbResult.M_MethodResult(MC_Reset,lastResult,ADR(_lastResult)) = FALSE THEN
	RETURN;
END_IF

IF _fbResult.P_MethodResult = E_Result.S_OK THEN
	_state := 0;
	fbMCReset(axis := axisRef,Execute := FALSE);
END_IF


_fbResult.P_MethodResult := E_Result.S_WORKING;

CASE _state OF
	0:
		fbMCReset(Axis := axisRef, Execute  := TRUE);
		_state := 1;
	1:
		fbMCReset(Axis := axisRef);	
		IF fbMCReset.Done = TRUE AND fbMCReset.Error = FALSE THEN
			_fbResult.P_MethodResult := E_Result.S_OK;
		ELSIF fbMCReset.Done = FALSE AND fbMCReset.Error = TRUE THEN 
			_fbResult.P_MethodResult := E_Result.S_FAILED;
		END_IF		
END_CASE
END_METHOD

METHOD PUBLIC MC_Stop : HResult
VAR_INPUT
	lastResult : HResult;
	Execute : BOOL;
	Deceleration : LREAL; 
	Jerk : LREAL;
END_VAR
VAR_OUTPUT
	Busy : BOOL;
	Active : BOOL;
	Error : BOOL;
	ErrorID : UDINT;	
END_VAR
VAR_INST
	_fbResult : FB_ResultHelper_V2_1;
	_lastResult : HResult;	
	_state : DINT;
END_VAR
IF _fbResult.M_MethodResult(MC_Stop,lastResult,ADR(_lastResult)) = FALSE THEN
	RETURN;
END_IF

IF _fbResult.P_MethodResult = E_Result.S_OK THEN
	_state := 0;
END_IF


_fbResult.P_MethodResult := E_Result.S_WORKING;

CASE _state OF
	0:
		fbMCStop(Axis := axisRef, Execute  := Execute ,Deceleration := Deceleration,Jerk := Jerk);
		IF fbMCStop.Done = TRUE AND fbMCStop.Error = FALSE THEN
			_fbResult.P_MethodResult := E_Result.S_OK;
		ELSIF fbMCStop.Done = FALSE AND fbMCStop.Error = TRUE THEN 
			_fbResult.P_MethodResult := E_Result.S_FAILED;
		END_IF		
END_CASE
END_METHOD

END_FUNCTION_BLOCK

// ---- FBs/FB_Kinenmatics_V2.TcPOU
FUNCTION_BLOCK FB_Kinenmatics_V2
VAR_INPUT
	intialVelocity : LREAL;
	intialPosition : LREAL;
	intialAcceleration : LREAL;
	intialJerk : LREAL;
	jerkLimit : LREAL;
	accelLimit : LREAL;
	decelLimit : LREAL;
	velocityLimit : LREAL;
	positionDelta : LREAL;
	timeToComplete : LREAL;
	discriment : LREAL;
END_VAR
VAR_OUTPUT
	minTime : LREAL;
	velocityOutput : LREAL;
	accelOutput : LREAL;
	jerkOutput : LREAL;
	error : BOOL;
	errorMsg : STRING;	
END_VAR
VAR
	positionMid : LREAL;
	positionQuarter : LREAL;
	//Caculating max values for a Jerk limited move
	jerkMoveAccelMax : LREAL;
	jerkMoveTimeToMaxAccel : LREAL;
	jerkMoveVelocityAtMaxAccel : LREAL;	
	jerkMoveVelocityMax : LREAL;
	jerkMoveTimeToMaxVelocity : LREAL;
	jerkMoveTimeToCompleteMin : LREAL;
	jerkMoveJerkLimitForTargetTime : LREAL;
	
	accelMoveTimeToMaxAccel : LREAL;
	accelMoveMaxVelocity : LREAL;
	accelMoveTimeForAccelConstantMove : LREAL;
	accelMoveTimeToCompleteMove : LREAL;

	accelMoveNewMaxAccel: LREAL;

	accelVelocityMoveTimeToMaxVelocity : LREAL;	
	accelVelocityMoveTimeFromMaxVelocityToMidPoint : LREAL;	
	accelVelocityTimeToCompleteMove : LREAL;

	


END_VAR

VAR
	jerkSegment : ARRAY [0..6] OF LREAL;
	accelSegment : ARRAY [0..6] OF LREAL;
	velocitySegment	: ARRAY [0..6] OF LREAL;
	positionSegment : ARRAY [0..6] OF LREAL;
	timeSegmentDelta : ARRAY [0..6] OF LREAL;
	timeSegment : ARRAY [0..6] OF TIME;	
	a : LREAL;
	b : LREAL;
	c : LREAL;	
	
	state : DINT;
	jerkLimitToAccelLimit : LREAL;
	timeToCompleteMinAccelMove : LREAL; 
END_VAR

IF positionDelta <= 0 OR timeToComplete <= 0 OR accelLimit <= 0 OR decelLimit <= 0 OR velocityLimit <= 0 OR jerkLimit <= 0 THEN
	RETURN;
END_IF

positionMid := positionDelta/2.0;
positionQuarter := positionDelta/4.0;
accelOutput := accelLimit;
jerkOutput := jerkLimit;
velocityOutput := velocityLimit;

state := M_JerkLimitedMove(positionDelta,
	jerkLimit,
	accelLimit,
	decelLimit,
	velocityLimit,
	timeToComplete,
	jerkOutput => jerkOutput,
	timeToCompleteMin => minTime,
	jerkLimitToAccelLimit => jerkLimitToAccelLimit,
	timeToCompleteMinAccelMove => timeToCompleteMinAccelMove,
	error => error,
	errorMsg => errorMsg
);
IF state = 1 THEN
	state := M_AccelLimitedMove(positionDelta,
		jerkLimit,
		accelLimit,
		decelLimit,
		velocityLimit,
		timeToComplete,
		jerkLimitToAccelLimit := jerkLimitToAccelLimit,
		timeToCompleteMinAccelMove := timeToCompleteMinAccelMove,
		jerkOutput => jerkOutput,
		accelOutput => accelOutput,
		error => error,
		errorMsg => errorMsg
	);
END_IF

RETURN;












(*
//Solve for t jerk limited equation positionMid = jerkLimit * t^3, 
//t = (positionMid/jerkLimit) ^(1/3) where t = 1/4 of the time to complete the move
jerkMoveTimeToMaxAccel := EXPT(positionMid/jerkLimit,1.0/3.0);
jerkMoveAccelMax := jerkLimit * jerkMoveTimeToMaxAccel;
jerkMoveVelocityAtMaxAccel := jerkMoveTimeToMaxAccel * jerkMoveAccelMax;
jerkMoveTimeToCompleteMin := jerkMoveTimeToMaxAccel * 4.0;

IF jerkMoveTimeToCompleteMin > timeToComplete THEN
	minTime := jerkMoveTimeToCompleteMin;
	errorMsg := 'Jerk limit too low';
	error := TRUE;			
	RETURN;
ELSE
	errorMsg := '';	
	error := FALSE;			
END_IF

IF (accelLimit < jerkMoveAccelMax) OR velocityLimit <= jerkMoveVelocityAtMaxAccel THEN
	//Caculate known values
	accelMoveTimeToMaxAccel := accelLimit/jerkLimit;
	positionSegment[0] := 1.0/6.0 * jerkLimit * EXPT(accelMoveTimeToMaxAccel,3.0);
	velocitySegment[0] := 0.5 * jerkLimit * EXPT(accelMoveTimeToMaxAccel,2.0) + intialVelocity;
	accelSegment[0] := jerkLimit*accelMoveTimeToMaxAccel;
	
	//set up quardatic formula 
	// 1/2*accelLimit*t^2 + (velocitySegment[0] + (accelLimit[0]*accelMoveTimeToMaxAccel)*t + (velocitySegment[0] * accelMoveTimeToMaxAccel)+accelSegment[0]*0.5*accelMoveTimeToMaxAccel^2
	a := 0.5 * accelSegment[0];
	b :=  velocitySegment[0] + accelSegment[0]*accelMoveTimeToMaxAccel;
	c := ((velocitySegment[0] * accelMoveTimeToMaxAccel)+accelSegment[0]*0.5*EXPT(accelMoveTimeToMaxAccel,2.0)) - positionMid;
	
	//Make sure discriment > 0 otherwise program will crash
	discriment := (EXPT(b,2.0) - 4.0 * a *c);
	IF discriment > 0 THEN
		accelMoveTimeForAccelConstantMove := (-b + EXPT(EXPT(b,2.0) -4.0 * a *c,0.5))/(2*a); //solve for quadtratic
		accelMoveTimeToCompleteMove := 2.0*(accelMoveTimeToMaxAccel * 2.0 + accelMoveTimeForAccelConstantMove); // This value is the fastest the machine can move with the accel limit
		accelMoveMaxVelocity := accelMoveTimeToCompleteMove/2*accelSegment[0]-EXPT(accelSegment[0],2.0)/jerkLimit;
		IF accelMoveMaxVelocity > velocityLimit THEN
			accelVelocityMoveTimeToMaxVelocity := velocityLimit/accelLimit + accelLimit/(jerkLimit);
			positionSegment[1] := velocitySegment[0]*(accelVelocityMoveTimeToMaxVelocity-2.0*accelMoveTimeToMaxAccel) + 0.5*accelLimit*EXPT((accelVelocityMoveTimeToMaxVelocity-2.0*accelMoveTimeToMaxAccel),2.0);
			velocitySegment[1] := velocitySegment[0] + accelLimit * (accelVelocityMoveTimeToMaxVelocity-2.0*accelMoveTimeToMaxAccel);
			positionSegment[2] := velocitySegment[1] * accelMoveTimeToMaxAccel +  0.5*accelLimit*EXPT((accelMoveTimeToMaxAccel),2.0) - 1.0/6.0 * jerkLimit * EXPT(accelMoveTimeToMaxAccel,3.0);
			//positionSegment[0] :=velocitySegment[0]*(accelVelocityMoveTimeToMaxVelocity-2.0*accelMoveTimeToMaxAccel);
			positionSegment[3] := positionMid - (positionSegment[0] + positionSegment[1] + positionSegment[2]);
			accelVelocityMoveTimeFromMaxVelocityToMidPoint := positionSegment[3]/velocityLimit;
			accelVelocityTimeToCompleteMove := 2.0*(accelVelocityMoveTimeToMaxVelocity + accelVelocityMoveTimeFromMaxVelocityToMidPoint);
			IF	accelVelocityTimeToCompleteMove < timeToComplete THEN
				errorMsg := '';		
				error := FALSE;						
				a := 1/jerkLimit;
				b := -(accelVelocityMoveTimeToMaxVelocity + timeToComplete - accelVelocityTimeToCompleteMove); //-timeToComplete/2.0; //
				c := velocityLimit;
				discriment := (EXPT(b,2.0) - 4.0 * a *c);
				IF discriment > 0 THEN
					minTime := accelVelocityTimeToCompleteMove;
					velocityOutput := velocityLimit;
					accelOutput := (-b - EXPT(EXPT(b,2.0) -4.0 * a *c,0.5))/(2*a);
					jerkOutput := jerkLimit; 
				END_IF	
			ELSIF accelVelocityTimeToCompleteMove > timeToComplete THEN
				minTime := accelVelocityTimeToCompleteMove;				
				errorMsg := 'velocity limit to low';	
				error := TRUE;		
				RETURN;	
			ELSIF accelVelocityTimeToCompleteMove = timeToComplete THEN
				minTime := accelVelocityTimeToCompleteMove;
				velocityOutput := velocityLimit;
				accelOutput := accelLimit;
				jerkOutput := jerkLimit; 			
			END_IF
		ELSIF accelMoveTimeToCompleteMove > timeToComplete THEN 
				minTime := accelMoveTimeToCompleteMove;			
			errorMsg := 'accel limit to low';
			error := TRUE;
			RETURN;
		ELSIF accelMoveTimeToCompleteMove < timeToComplete THEN
			minTime := accelMoveTimeToCompleteMove;
			error := FALSE;			
			errorMsg := '';	
			//Vmax = t*a-a^2/(2*j) positionMid = Intergrate(Vmax) = timeToCompleteMove/(4.0 * jerkLimit)*a^2 + ((timeToCompleteMove/2)^2)/2; solve with quaddratic
			a := -(timeToComplete/(4.0*jerkLimit));
			b := EXPT(timeToComplete/2.0,2.0)/2.0;
			c := -positionMid;			
			discriment := (EXPT(b,2.0) - 4.0 * a *c);
			IF discriment > 0 THEN
				accelOutput := (-b + EXPT(EXPT(b,2.0) -4.0 * a *c,0.5))/(2*a); //solve for quadtratic
			END_IF
			jerkOutput := jerkLimit;
			velocityOutput := velocityLimit;			
		ELSE
			error := FALSE;					
			errorMsg := '';	
		END_IF	
	END_IF
	//RETURN; // accel limited only
ELSIF accelLimit < jerkMoveAccelMax AND velocityLimit < jerkMoveVelocityAtMaxAccel THEN
	RETURN; // accel limited only and might be velocity limited
ELSIF accelLimit >= jerkMoveAccelMax AND velocityLimit >= jerkMoveVelocityAtMaxAccel THEN
	//jerkLimit = positionMid/(timeToComplete/4)^(3)
	minTime := jerkMoveTimeToCompleteMin;
	jerkMoveJerkLimitForTargetTime := positionMid/EXPT(timeToComplete/4,3.0);
	jerkOutput := jerkMoveJerkLimitForTargetTime;
	velocityOutput := velocityLimit;
	accelOutput := accelLimit;
	RETURN; // jerk limited
END_IF
	


// Max velocity in a jerk only limited move = positionMid = 1/2 * jerkLimit * t^2
// jerkMoveTimeToMaxVelocity := EXPT(positionMid*6/jerkLimit,1.0/3.0);
// jerkMoveVelocityMax := 1.0/2.0 * jerkLimit * EXPT(jerkMoveTimeToMaxVelocity,2);


*)

METHOD PROTECTED M_AccelLimitedMove : DINT
VAR_INPUT
	position : LREAL;
	jerkLimit : LREAL;
	accelLimit : LREAL;
	decelLimit : LREAL;
	velocityLimit : LREAL;
	timeToComplete : LREAL;
	jerkLimitToAccelLimit : LREAL;
	timeToCompleteMinAccelMove : LREAL;
END_VAR
VAR_OUTPUT
	jerkOutput : LREAL;
	accelOutput : LREAL;
	timeToCompleteMin : LREAL;	
	error : BOOL;
	errorMsg : STRING;	
END_VAR
VAR
	positionMid : LREAL;
	timeToMaxAccel : LREAL;
	minJerkToAccelLimitMove : LREAL;
	accelMax : LREAL;
	velocityMax : LREAL;
	a : LREAL;	
	b : LREAL;
	c : LREAL;
	timeToAccelMaxMoveMin : LREAL;
	x : DINT;
END_VAR
VAR_INST

	jerkAdjustment : LREAL;

	whatsMyValue : LREAL;
	autoCounter : BOOL;
	rateOfChange : LREAL := 1;
	slopCaculation : LREAL;
	jerkStep : LREAL;
END_VAR
positionMid := position/2.0;

timeToAccelMaxMoveMin := accelLimit/jerkLimitToAccelLimit;
//Accel limit hit before jerk limit hit in a jerk limited move. 

IF jerkLimitToAccelLimit > 0 THEN //Might make a function
	jerkStep := (jerkLimit - jerkLimitToAccelLimit)/10.0;
	jerkAdjustment := jerkLimitToAccelLimit + jerkStep;
	timeToMaxAccel := accelLimit/jerkAdjustment;	
 	FOR x := 0 TO 8 BY 1 DO // can't find a soultion with an equation so increasing jerk slowly and finding a min value thats greater than target. 
		timeSegmentDelta[0] := timeToMaxAccel;
		jerkSegment[0] := jerkAdjustment;
		jerkSegment[1] := 0;
		jerkSegment[2] := -jerkAdjustment;
		jerkSegment[3] := -jerkAdjustment;
		jerkSegment[4] := 0;
		jerkSegment[5] := jerkAdjustment;	
		M_SegmentCaculator();
	(*
	a = 1/2*accelLimit*t^2 + 
	b = (velocitySegment[0] + (accelSegment[0]*accelMoveTimeToMaxAccel)*t +
	c = (velocitySegment[0] * accelMoveTimeToMaxAccel)+accelSegment[0]*0.5*accelMoveTimeToMaxAccel^2
	*)	
		//find time where accel is a constant
		M_QuadraticEquation(
			a := 0.5*accelLimit, 
			b := velocitySegment[0] + (accelLimit*timeSegmentDelta[0]),
			c := (velocitySegment[0] * timeSegmentDelta[0])+accelSegment[0]*0.5*EXPT(timeSegmentDelta[0],2.0) - positionMid,
			plusResult => timeSegmentDelta[1]);
		//Caculate the rest of the time segments	
		timeSegmentDelta[2] := timeSegmentDelta[0];
		timeSegmentDelta[3] := timeSegmentDelta[0];
		timeSegmentDelta[4] := timeSegmentDelta[1];
		timeSegmentDelta[5] := timeSegmentDelta[0];	
		timeToCompleteMin := timeSegmentDelta[0] + timeSegmentDelta[1] + timeSegmentDelta[2] + timeSegmentDelta[3] + timeSegmentDelta[4] + timeSegmentDelta[5];
		IF timeToCompleteMin <= timeToComplete THEN
			jerkOutput := jerkAdjustment; 
			EXIT;	
		ELSE	
			jerkAdjustment := jerkAdjustment + jerkStep;
		END_IF
	END_FOR
	
	IF timeToCompleteMin < timeToComplete THEN
		//Vmax = t*a-a^2/(2*j) positionMid = Integrate(Vmax) = timeToCompleteMove/(4.0 * jerkLimit)*a^2 + ((timeToCompleteMove/2)^2)/2; solve with quaddratic
		M_QuadraticEquation(
			a := -(timeToComplete)/(4.0*jerkAdjustment),
			b := EXPT(timeToComplete/2.0,2.0)/2.0,
			c := -positionMid,
			plusResult => accelOutput);		
	END_IF
	M_SegmentCaculator();
ELSE
	IF timeToCompleteMin < timeToComplete THEN
		//Vmax = t*a-a^2/(2*j) positionMid = Intergrate(Vmax) = timeToCompleteMove/(4.0 * jerkLimit)*a^2 + ((timeToCompleteMove/2)^2)/2; solve with quaddratic
		M_QuadraticEquation(
			a := -(timeToComplete)/(4.0*jerkLimit),
			b := EXPT(timeToComplete/2.0,2.0)/2.0,
			c := -positionMid,
			plusResult => accelOutput);		
	END_IF
	M_SegmentCaculator();	
END_IF
END_METHOD

METHOD PROTECTED M_AccelVelocityLimitedMove : LREAL
VAR_INPUT
END_VAR
END_METHOD

METHOD PROTECTED M_JerkLimitedMove : DINT
VAR_INPUT
	position : LREAL;
	jerkLimit : LREAL;
	accelLimit : LREAL;
	decelLimit : LREAL;
	velocityLimit : LREAL;
	timeToComplete : LREAL;
END_VAR
VAR_OUTPUT
	jerkOutput : LREAL;
	jerkLimitToAccelLimit : LREAL;
	timeToCompleteMin : LREAL;
	timeToCompleteMinAccelMove : LREAL;
	error : BOOL;
	errorMsg : STRING;	
END_VAR
VAR
	positionMid : LREAL;
	timeToMaxAccel : LREAL;
	accelMax : LREAL;
	velocityMax : LREAL;
	jerkLimitedByAccel: BOOL;
END_VAR
//Find mid position
positionMid := position/2.0;

//determine if accel limit limits jerk limited move
jerkLimitToAccelLimit := EXPT(EXPT(accelLimit,(3))/positionMid,0.5);

IF jerkLimitToAccelLimit < jerkLimit THEN
	jerkLimit := jerkLimitToAccelLimit;
	jerkLimitedByAccel := TRUE;
END_IF

//Find time to max accel with jerk limit
timeToMaxAccel := EXPT(positionMid/jerkLimit,1.0/3.0);

//Time to complete is timeToMaxAccel * 4
timeToCompleteMin := timeToMaxAccel * 4.0;

IF timeToComplete > timeToCompleteMin THEN
	jerkOutput := positionMid/EXPT(timeToComplete/4,3.0);	
	timeToMaxAccel := EXPT(positionMid/jerkOutput,1.0/3.0);	
END_IF


//Caculate max accel
accelMax := jerkOutput * timeToMaxAccel;



IF accelMax < accelLimit AND velocityMax < velocityLimit THEN
	timeSegmentDelta[0] := timeToMaxAccel;
	timeSegmentDelta[1] := timeToMaxAccel;
	timeSegmentDelta[2] := timeToMaxAccel;
	timeSegmentDelta[3] := timeToMaxAccel;
	timeSegmentDelta[4] := 0;
	timeSegmentDelta[5] := 0;
	timeSegmentDelta[6] := 0;
	
	jerkSegment[0] := jerkOutput;
	jerkSegment[1] := -jerkOutput;
	jerkSegment[2] := -jerkOutput;
	jerkSegment[3] := jerkOutput;	
	jerkSegment[4] := 0;		
	jerkSegment[5] := 0;	
	jerkSegment[6] := 0;	

	M_SegmentCaculator();
	
ELSIF accelMax > accelLimit THEN
	errorMsg := 'Accel limited move';	
	error := TRUE;
	M_JerkLimitedMove := 1;	
	RETURN;		
END_IF

IF timeToCompleteMin > timeToComplete AND jerkLimitedByAccel = FALSE THEN
	errorMsg := 'Jerk limit too low';
	error := TRUE;			
	RETURN;	
ELSIF timeToCompleteMin > timeToComplete AND jerkLimitedByAccel = TRUE THEN
	errorMsg := 'Accel limited move';	
	error := TRUE;	
	M_JerkLimitedMove := 1;	
	timeToCompleteMinAccelMove := timeToCompleteMin;
	RETURN;			
END_IF
END_METHOD

METHOD PROTECTED M_QuadraticEquation : LREAL
VAR_INPUT
	a : LREAL;
	b : LREAL;
	c : LREAL;	
END_VAR
VAR
	discriment : LREAL;
END_VAR	
VAR_OUTPUT
	error : BOOL;
	plusResult : LREAL;
	negResult : LREAL;
END_VAR
discriment := (EXPT(b,2.0) - 4.0 * a *c);
IF discriment >= 0 THEN
	M_QuadraticEquation := (-b + EXPT(EXPT(b,2.0) -4.0 * a *c,0.5))/(2*a);	
	plusResult := (-b + EXPT(EXPT(b,2.0) -4.0 * a *c,0.5))/(2*a);
	negResult := (-b - EXPT(EXPT(b,2.0) -4.0 * a *c,0.5))/(2*a);	
ELSE
	error := TRUE;
END_IF
END_METHOD

METHOD PROTECTED M_SegmentCaculator : BOOL
VAR_INPUT
END_VAR

VAR
	x: INT;
	y: INT;
END_VAR
//This caculates each segment of the move. First are intial which are always 0; 
timeSegment[0] := TO_TIME(timeSegmentDelta[0]*1000);
accelSegment[0] :=  intialAcceleration + jerkSegment[0] * timeSegmentDelta[0];
velocitySegment[0] := intialVelocity + intialAcceleration * timeSegmentDelta[0] + 1.0/2.0*jerkSegment[0]*EXPT(timeSegmentDelta[0],2.0);
positionSegment[0] := intialPosition + intialVelocity * timeSegmentDelta[0] + 1.0/2.0 * intialAcceleration * EXPT(timeSegmentDelta[0],2.0) + 1.0/6.0*jerkSegment[0]*EXPT(timeSegmentDelta[0],3.0);
	
FOR x := 1 TO 6 BY 1 DO
	y := x-1;
	timeSegment[x] := timeSegment[y] + TO_TIME(timeSegmentDelta[x]*1000);
	
	accelSegment[x] := accelSegment[y] + jerkSegment[x] * timeSegmentDelta[x];			
	
	velocitySegment[x] := velocitySegment[y] + accelSegment[y] * timeSegmentDelta[x] + 1.0/2.0*jerkSegment[x]*EXPT(timeSegmentDelta[x],2.0);	

	positionSegment[x] := positionSegment[y] + velocitySegment[y] * timeSegmentDelta[x] + 1.0/2.0 * accelSegment[y] * EXPT(timeSegmentDelta[x],2.0) + 1.0/6.0*jerkSegment[x]*EXPT(timeSegmentDelta[x],3.0);

END_FOR
END_METHOD

END_FUNCTION_BLOCK

// ---- FBs/System/FB_ConfigControl.TcPOU
FUNCTION_BLOCK FB_ConfigControl
VAR_INPUT
	a_pFBConfigJson : POINTER TO POINTER TO FB_ConfigBase; //pointer to pointer is an array
	ua_pFBConfigJson : UDINT;
END_VAR
VAR_OUTPUT
END_VAR
VAR
	fbRecipeJson : FB_ValuesJson;
	fbSystemJson : FB_ValuesJson;
	fbIOJson : FB_ValuesJson;
	fbAxisJson : FB_NCAxisJson_V2;
END_VAR

METHOD PUBLIC M_GetJsonAxis : HResult
VAR_INPUT
	lastResult : HRESULT;
END_VAR
VAR_IN_OUT
	pDoc : STRING(50000);
END_VAR
VAR CONSTANT
	uSizeOfStAnyType : UDINT := SIZEOF(PVOID);
END_VAR
VAR_INST
	uSizeOfArray : DINT;
	x : DINT;
	pFBConfigJson : POINTER TO POINTER TO FB_ConfigBase;	
	_fbResult : FB_ResultHelper_V2;
	pResult : POINTER TO HRESULT;
END_VAR
IF _fbResult.M_MethodResult(M_GetJsonAxis,ADR(pResult),lastResult) = FALSE THEN
	RETURN;
END_IF

uSizeOfArray := ua_pFBConfigJson/uSizeOfStAnyType - 1; //get number of items in array

fbAxisJson.ParseDocument(pDoc);
fbAxisJson.M_PraseSchemaJson();
FOR x := 0 TO uSizeOfArray BY 1 DO
	pFBConfigJson := a_pFBConfigJson + uSizeOfStAnyType*x;
	lastResult := pFBConfigJson^^.F_AXIS(lastResult,fbAxisJson.P_sJsonValues.jsonValue,ADR(fbAxisJson),TRUE);
END_FOR

fbAxisJson.CopyDocument(pDoc,SIZEOF(pDoc));
END_METHOD

METHOD PUBLIC M_GetJsonIO : HResult
VAR_INPUT
	lastResult : HRESULT;
END_VAR
VAR_IN_OUT
	pDoc : STRING(50000);
END_VAR
VAR CONSTANT
	uSizeOfStAnyType : UDINT := SIZEOF(PVOID);
END_VAR
VAR_INST
	uSizeOfArray : DINT;
	x : DINT;
	pFBConfigJson : POINTER TO POINTER TO FB_ConfigBase;	
	_fbResult : FB_ResultHelper_V2;
	pResult : POINTER TO HRESULT;
END_VAR
IF _fbResult.M_MethodResult(M_GetJsonIO,ADR(pResult),lastResult) = FALSE THEN
	RETURN;
END_IF


uSizeOfArray := ua_pFBConfigJson/uSizeOfStAnyType - 1; //get number of items in array


fbIOJson.M_CreateSchemaJson();
FOR x := 0 TO uSizeOfArray BY 1 DO
	pFBConfigJson := a_pFBConfigJson + uSizeOfStAnyType*x;
	lastResult := pFBConfigJson^^.F_IO(lastResult,fbIOJson.P_sJsonValues.jsonValue,ADR(fbIOJson),FALSE);
END_FOR


fbIOJson.CopyDocument(pDoc,SIZEOF(pDoc));
END_METHOD

METHOD PUBLIC M_GetJsonRecipe : HResult
VAR_INPUT
	lastResult : HRESULT;
END_VAR
VAR_IN_OUT
	pDoc : STRING(10000);
END_VAR

VAR CONSTANT
	uSizeOfStAnyType : UDINT := SIZEOF(PVOID);
END_VAR

VAR_INST
	bGet : BOOL;
	uSizeOfArray : DINT;
	x : DINT;
	pFBConfigJson : POINTER TO POINTER TO FB_ConfigBase;	
	_fbResult : FB_ResultHelper_V2;
	pResult : POINTER TO HRESULT;
END_VAR
IF _fbResult.M_MethodResult(M_GetJsonRecipe,ADR(pResult),lastResult) = FALSE THEN
	RETURN;
END_IF

uSizeOfArray := ua_pFBConfigJson/uSizeOfStAnyType - 1; //get number of items in array

fbRecipeJson.M_PraseSchemaJson();
FOR x := 0 TO uSizeOfArray BY 1 DO
	pFBConfigJson := a_pFBConfigJson + uSizeOfStAnyType*x;
	lastResult := pFBConfigJson^^.F_Recipe(lastResult,fbRecipeJson.P_sJsonValues.jsonValue,ADR(fbRecipeJson),TRUE);
END_FOR

fbRecipeJson.CopyDocument(pDoc,SIZEOF(pDoc));
END_METHOD

METHOD PUBLIC M_GetJsonSystem : HResult
VAR_INPUT
	lastResult : HRESULT;
END_VAR
VAR_IN_OUT
	pDoc : STRING(50000);
END_VAR
VAR CONSTANT
	uSizeOfStAnyType : UDINT := SIZEOF(PVOID);
END_VAR
VAR_INST
	uSizeOfArray : DINT;
	x : DINT;
	pFBConfigJson : POINTER TO POINTER TO FB_ConfigBase;	
	_fbResult : FB_ResultHelper_V2;
	pResult : POINTER TO HRESULT;
END_VAR
IF _fbResult.M_MethodResult(M_GetJsonSystem,ADR(pResult),lastResult) = FALSE THEN
	RETURN;
END_IF

uSizeOfArray := ua_pFBConfigJson/uSizeOfStAnyType - 1; //get number of items in array


fbSystemJson.M_CreateSchemaJson();
FOR x := 0 TO uSizeOfArray BY 1 DO
	pFBConfigJson := a_pFBConfigJson + uSizeOfStAnyType*x;
	lastResult := pFBConfigJson^^.F_System(lastResult,fbSystemJson.P_sJsonValues.jsonValue,ADR(fbSystemJson),TRUE);
END_FOR

fbSystemJson.CopyDocument(pDoc,SIZEOF(pDoc));
END_METHOD

METHOD PUBLIC M_SetJsonAxis : HResult
VAR_INPUT
	lastResult : HRESULT;
END_VAR
VAR_IN_OUT
	pDoc : STRING(50000);
END_VAR
VAR CONSTANT
	uSizeOfStAnyType : UDINT := SIZEOF(PVOID);
END_VAR
VAR_INST
	uSizeOfArray : DINT;
	x : DINT;
	pFBConfigJson : POINTER TO POINTER TO FB_ConfigBase;	
	_fbResult : FB_ResultHelper_V2;
	pResult : POINTER TO HRESULT;
END_VAR
IF _fbResult.M_MethodResult(M_SetJsonAxis,ADR(pResult),lastResult) = FALSE THEN
	RETURN;
END_IF

uSizeOfArray := ua_pFBConfigJson/uSizeOfStAnyType - 1; //get number of items in array


fbAxisJson.M_CreateSchemaJson();
FOR x := 0 TO uSizeOfArray BY 1 DO
	pFBConfigJson := a_pFBConfigJson + uSizeOfStAnyType*x;
	lastResult := pFBConfigJson^^.F_AXIS(lastResult,fbAxisJson.P_sJsonValues.jsonValue,ADR(fbAxisJson),TRUE);
END_FOR

fbAxisJson.CopyDocument(pDoc,SIZEOF(pDoc));
END_METHOD

METHOD PUBLIC M_SetJsonIO : HResult
VAR_INPUT
	lastResult : HRESULT;
END_VAR
VAR_IN_OUT
	pDoc : STRING(50000);
END_VAR
VAR CONSTANT
	uSizeOfStAnyType : UDINT := SIZEOF(PVOID);
END_VAR
VAR_INST
	uSizeOfArray : DINT;
	x : DINT;
	pFBConfigJson : POINTER TO POINTER TO FB_ConfigBase;	
	_fbResult : FB_ResultHelper_V2;
	pResult : POINTER TO HRESULT;
END_VAR
IF _fbResult.M_MethodResult(M_SetJsonIO,ADR(pResult),lastResult) = FALSE THEN
	RETURN;
END_IF

uSizeOfArray := ua_pFBConfigJson/uSizeOfStAnyType - 1; //get number of items in array


fbIOJson.M_CreateSchemaJson();
FOR x := 0 TO uSizeOfArray BY 1 DO
	pFBConfigJson := a_pFBConfigJson + uSizeOfStAnyType*x;
	lastResult := pFBConfigJson^^.F_IO(lastResult,fbIOJson.P_sJsonValues.jsonValue,ADR(fbIOJson),TRUE);
END_FOR


fbIOJson.CopyDocument(pDoc,SIZEOF(pDoc));
END_METHOD

METHOD PUBLIC M_SetJsonRecipe : HResult
VAR_INPUT
	lastResult : HRESULT;
END_VAR
VAR_IN_OUT
	pDoc : STRING(10000);
END_VAR

VAR CONSTANT
	uSizeOfStAnyType : UDINT := SIZEOF(PVOID);
END_VAR

VAR_INST
	bGet : BOOL;
	uSizeOfArray : DINT;
	x : DINT;
	pFBConfigJson : POINTER TO POINTER TO FB_ConfigBase;	
	_fbResult : FB_ResultHelper_V2;
	pResult : POINTER TO HRESULT;
END_VAR
IF _fbResult.M_MethodResult(M_SetJsonRecipe,ADR(pResult),lastResult) = FALSE THEN
	RETURN;
END_IF

uSizeOfArray := ua_pFBConfigJson/uSizeOfStAnyType - 1; //get number of items in array

fbRecipeJson.M_CreateSchemaJson();
FOR x := 0 TO uSizeOfArray BY 1 DO
	pFBConfigJson := a_pFBConfigJson + uSizeOfStAnyType*x;
	lastResult := pFBConfigJson^^.F_Recipe(lastResult,fbRecipeJson.P_sJsonValues.jsonValue,ADR(fbRecipeJson),FALSE);
END_FOR

fbRecipeJson.CopyDocument(pDoc,SIZEOF(pDoc));
END_METHOD

METHOD PUBLIC M_SetJsonSystem : HResult
VAR_INPUT
	lastResult : HRESULT;
END_VAR
VAR_IN_OUT
	pDoc : STRING(50000);
END_VAR
VAR CONSTANT
	uSizeOfStAnyType : UDINT := SIZEOF(PVOID);
END_VAR
VAR_INST
	uSizeOfArray : DINT;
	x : DINT;
	pFBConfigJson : POINTER TO POINTER TO FB_ConfigBase;	
	_fbResult : FB_ResultHelper_V2;
	pResult : POINTER TO HRESULT;
END_VAR
IF _fbResult.M_MethodResult(M_SetJsonSystem,ADR(pResult),lastResult) = FALSE THEN
	RETURN;
END_IF

uSizeOfArray := ua_pFBConfigJson/uSizeOfStAnyType - 1; //get number of items in array


fbSystemJson.M_CreateSchemaJson();
FOR x := 0 TO uSizeOfArray BY 1 DO
	pFBConfigJson := a_pFBConfigJson + uSizeOfStAnyType*x;
	lastResult := pFBConfigJson^^.F_System(lastResult,fbSystemJson.P_sJsonValues.jsonValue,ADR(fbSystemJson),FALSE);
END_FOR


fbSystemJson.CopyDocument(pDoc,SIZEOF(pDoc));
END_METHOD

END_FUNCTION_BLOCK

// ---- FBs/JSON/FB_ValuesJson.TcPOU
FUNCTION_BLOCK FB_ValuesJson EXTENDS FB_JsonSchemaEx_OLD
VAR_INPUT
END_VAR
VAR_OUTPUT
	P_sJsonid			: MPM_JsonParser.DUT_JsonSchema := (member := '_id', typeClass := E_TypeClassEx.TYPE_STRING,jsonValueRoot := jsonRoot);
	P_sJsonTimeStamp	: MPM_JsonParser.DUT_JsonSchema := (member := 'time_stamp', typeClass := E_TypeClassEx.TYPE_FILETIME,jsonValueRoot := jsonRoot);		
	P_sJsonValues		: MPM_JsonParser.DUT_JsonSchema := (member := 'values', typeClass := E_TypeClassEx.TYPE_JSON,jsonValueRoot := jsonRoot);
END_VAR
VAR
	jsonRoot : SJsonValue;	
END_VAR

METHOD PUBLIC  M_CreateSchemaJson : BOOL
VAR_IN_OUT
END_VAR
VAR
	
END_VAR
jsonRoot := THIS^.NewDocument();
M_SetJsonSchema(jsonRoot,P_sJsonid);
M_SetJsonSchema(jsonRoot,P_sJsonValues);
M_SetJsonSchema(jsonRoot,P_sJsonTimeStamp);
END_METHOD

METHOD PUBLIC  M_PraseSchemaJson : BOOL
VAR_INPUT
END_VAR
jsonRoot := THIS^.GetDocumentRoot();
IF jsonRoot > 0 THEN
	M_PraseJsonSchema(jsonRoot,P_sJsonid);
	M_PraseJsonSchema(jsonRoot,P_sJsonValues);
	M_PraseJsonSchema(jsonRoot,P_sJsonTimeStamp);
END_IF
END_METHOD

END_FUNCTION_BLOCK

// ---- FBs/Main/FB_PackMLControl_Auto.TcPOU
FUNCTION_BLOCK FB_PackMLControl_Auto EXTENDS FB_PackMLControl
VAR_INPUT
	ap_fbEvents : POINTER TO ARRAY [0..1023] OF POINTER TO FB_DiscreteEvents;	
END_VAR
VAR_OUTPUT
END_VAR
VAR
	state : E_PackMLStates := E_PackMLStates.idle;
	ap_fbEventsIdle : ARRAY [0..0] OF POINTER TO FB_DiscreteEvents;		
	ap_fbEventsStarting : ARRAY [0..0] OF POINTER TO FB_DiscreteEvents;		
	ap_fbEventsExecute : ARRAY [0..0] OF POINTER TO FB_DiscreteEvents;	
	ap_fbEventsStop : ARRAY [0..254] OF POINTER TO FB_DiscreteEvents;			
END_VAR

METHOD PROTECTED _mapping : HResult
VAR_INPUT
END_VAR
ap_fbEventsIdle[0] := ap_fbEvents^[0];
ap_fbEventsStarting[0] := ap_fbEvents^[1];
ap_fbEventsExecute[0] := ap_fbEvents^[5];
END_METHOD

METHOD PUBLIC M_Aborted : HResult
VAR_INPUT
END_VAR
END_METHOD

METHOD PUBLIC M_Aborting : HResult
VAR_INPUT
END_VAR
END_METHOD

METHOD PUBLIC M_Complete : HResult
VAR_INPUT
	lastResult : HResult;
END_VAR
VAR_OUTPUT
	abort : BOOL;
END_VAR
VAR_INST
	_fbResult : FB_ResultHelper_V2_1;	
	_lastResult : HRESULT;
	_state : POINTER TO DINT;
END_VAR
_state := ADR(state_complete);
IF _fbResult.M_MethodResult(M_Complete,lastResult,ADR(_lastResult)) = FALSE THEN
	RETURN;
END_IF

IF _fbResult.P_MethodResult = E_Result.S_OK THEN
	_state^ := 0;
END_IF

_fbResult.P_MethodResult := MPM_FBResult.E_Result.S_OK;
END_METHOD

METHOD PUBLIC M_Completing : HREsult
VAR_INPUT
	lastResult : HResult;
END_VAR
VAR_OUTPUT
	abort : BOOL;	
	stop : BOOL;
END_VAR
VAR_INST
	_fbResult : FB_ResultHelper_V2_1;	
	_lastResult : HRESULT;
	_state : POINTER TO DINT;
END_VAR
_state := ADR(state_completing);
IF _fbResult.M_MethodResult(M_Completing,lastResult,ADR(_lastResult)) = FALSE THEN
	RETURN;
END_IF

IF _fbResult.P_MethodResult = E_Result.S_OK THEN
	_state^ := 0;
END_IF

_fbResult.P_MethodResult := MPM_FBResult.E_Result.S_OK;
END_METHOD

METHOD PUBLIC M_Execute : HResult
VAR_INPUT
	lastResult : HResult;
END_VAR
VAR_OUTPUT
	stop : BOOL;
	suspend : BOOL;
	hold : BOOL;
END_VAR
VAR_INST
	_fbResult : FB_ResultHelper_V2_1;	
	_lastResult : HRESULT;
	_state : POINTER TO DINT;
	_ap_fbEventsExecute0_Result : HResult;
	_ap_fbEventsExecute1_Result : HResult;	
END_VAR
_state := ADR(state_execute);
IF _fbResult.M_MethodResult(M_Execute,lastResult,ADR(_lastResult)) = FALSE THEN
	RETURN;
END_IF

IF _fbResult.P_MethodResult = E_Result.S_OK THEN
	_state^ := 0;
END_IF

